// TIA Portal project "DrMartens2024_12_10_LMQTT_Client_V17" (V17)

(* hardware
DEVICE "S7-1200 station_1"  S7-1200 Station
   slot 0: "Rack_0"  S7-1200 Rack  Rack  V1.0
   slot 1: "MqttPlc1200"  CPU 1214C DC/DC/DC  6ES7 214-1AG40-0XB0  V4.4
DEVICE "S71500/ET200MP station_2"  S7-1500 station
   slot 0: "Rail_0"  Rack  6ES7 590-1***0-0AA0
   slot 1: "MqttPlc1500"  CPU 1517F-3 PN/DP  6ES7 517-3FP00-0AB0  V2.8
      slot 3: "CPU display_1"  6ES7591-1BA00-0AA0
      slot 32768: "PROFINET interface_1"  X1
         slot 32769: "Port_1"  X1 P1
         slot 32770: "Port_2"  X1 P2
      slot 33024: "PROFINET interface_2"  X2
      slot 33280: "DP interface_1"  X3
      slot 34817: "Virtual CP interface port_1"  Virtual CP interface port  Virtual CP interface port
*)

// ===== PLC "MqttPlc1200"  CPU 1214C DC/DC/DC =====

VAR_GLOBAL   // PLC tag table "Default tag table"
   "I0_0_Speed" AT %I0.0 : Bool;   // Speed - Sensor
   "I0_1_RunStop_Machine" AT %I0.1 : Bool;   // Relay
   "I0_2_Signal_Xilanh_Push" AT %I0.2 : Bool;   // Relay
   "I0_3_Signal_Pedal" AT %I0.3 : Bool;   // Relay: TRUE: Đi vào, FALSE : Đi ra
   "I0_4_RunStop_Inverter" AT %I0.4 : Bool;
   "I0_5_Spare" AT %I0.5 : Bool;
   "I0_6_Spare" AT %I0.6 : Bool;
   "I0_7_Spare" AT %I0.7 : Bool;
   "AI_Module_Ch00_Pressure_In" AT %IW96 : Int;   // Analog dòng
   "AI_Module_Ch01__Pressure_Out" AT %IW98 : Int;   // Analog spare
   "AI_Module_Ch02_Temperature" AT %IW100 : Int;   // Analog nhiệt độ
   "AI_Module_Ch03" AT %IW102 : Int;   // Analog Pressure Out
   "System_Byte" AT %MB1 : Byte;
   "FirstScan" AT %M1.0 : Bool;
   "DiagStatusUpdate" AT %M1.1 : Bool;
   "AlwaysTRUE" AT %M1.2 : Bool;
   "AlwaysFALSE" AT %M1.3 : Bool;
   "Clock_Byte" AT %MB0 : Byte;
   "Clock_10Hz" AT %M0.0 : Bool;
   "Clock_5Hz" AT %M0.1 : Bool;
   "Clock_2.5Hz" AT %M0.2 : Bool;
   "Clock_2Hz" AT %M0.3 : Bool;
   "Clock_1.25Hz" AT %M0.4 : Bool;
   "Clock_1Hz" AT %M0.5 : Bool;
   "Clock_0.625Hz" AT %M0.6 : Bool;
   "Clock_0.5Hz" AT %M0.7 : Bool;
   "M_Speed" AT %M100.0 : Bool;
   "M_RunStop_Machine" AT %M100.1 : Bool;
   "M_Xilanh_Push" AT %M100.2 : Bool;
   "M_Pedal" AT %M100.3 : Bool;
   "M_RunStop_Inverter" AT %M100.4 : Bool;
   "Input 5 Spare" AT %M100.5 : Bool;
   "Input 6 Spare" AT %M100.6 : Bool;
   "Input 7 Spare" AT %M100.7 : Bool;
   "M_Temperature" AT %MW4 : Int;
   "M_Current" AT %MW6 : Int;
   "M_AnalogPlc_Spare" AT %MW8 : Int;
   "M_Pressure Out" AT %MW16 : Int;
   "tag_idx" AT %MW18 : Int;
   "SignalP_RaisingCounter" AT %M200.0 : Bool;
   "SignalStatusMachineP" AT %M200.1 : Bool;
   "TagSignalStatusMachineP" AT %M200.2 : Bool;
   "TagSignalStatusMachineN" AT %M200.3 : Bool;
   "ClearDataBufferLossInShift" AT %M200.4 : Bool;
   "ClearDataBufferStatusMachineForServer" AT %M200.5 : Bool;
   "ClearSetDataDefaultLossGroupReason" AT %M200.6 : Bool;
   "PulseP_Check_ConnectHmi" AT %M200.7 : Bool;
   "Tag_1" AT %M500.0 : Bool;
   "Tag_2" AT %M601.0 : Bool;
   "Tag_3" AT %M601.2 : Bool;
   "Tag_4" AT %M600.4 : Bool;
   "Tag_5" AT %M700.0 : Bool;
   "Tag_6" AT %M700.1 : Bool;
   "Tag_7" AT %M700.2 : Bool;
   "AI_PLC_Ch00_Current" AT %IW64 : Int;   // AnalogPlcCh01
   "AI_PLC_Ch01" AT %IW66 : Int;   // AnalogPlcCh02
   "M_Pressure In" AT %MW20 : Int;
   "M_AnalogModule_Spare" AT %MW22 : Int;
   "Tag_8" AT %M201.0 : Bool;
   "Tag_9" AT %M202.1 : Bool;
   "Tag_10" AT %M303.0 : Bool;
   "Tag_11" AT %M303.2 : Bool;
   "Tag_12" AT %M303.1 : Bool;
   "Tag_13" AT %M404.0 : Bool;
   "Tag_14" AT %Q0.0 : Bool;
END_VAR

TYPE "SensorSimulation"
VERSION : 0.1
   STRUCT
      TimerTriggerON_x10ms : UInt := 100;   // Time-base x10ms
      TimerTriggerOFF_x10ms : UInt := 100;   // Time-base x10ms
      Output : Bool;
      nTempCounting : UInt;
   END_STRUCT;
END_TYPE

TYPE "DataShowChart"
VERSION : 0.1
   STRUCT
      Actual : DInt;
      Max : DInt;
      Min : DInt;
      AxisY_Max : DInt;
      AxisY_Min : DInt;
   END_STRUCT;
END_TYPE

TYPE "MachineEventDatatype"
VERSION : 0.1
   STRUCT
      id : UDInt;
      losscode : UInt;
      startTime : DTL;
      endTime : DTL;
      duration : UDInt;
      statusServer : USInt;   // 0: undefine; 1: stop; 2: run; 3: server-read; 4: server-updated
   END_STRUCT;
END_TYPE

TYPE "LossDescriptionDatatype"
VERSION : 0.1
   STRUCT
      description : String[30];
      group_id : UInt;
   END_STRUCT;
END_TYPE

TYPE "SpeedSensorType"
VERSION : 0.1
   STRUCT
      bStartCalculateSpeed : Bool;   // Bit lưu trạng thái vào quy trình đo speed
      TimeSpeed : Time;   // Time tính được giữa 2 lần interrupt
      idx : Int;   // Số lần tính speed
      "Out Current Speed" : Int;   // Tốc độ hiện tại đo được
   END_STRUCT;
END_TYPE

TYPE "AnalogSensorType"
VERSION : 0.1
   STRUCT
      MinRealScale : Real;   // 0V
      MaxRealScale : Real := 10.0;   // 10V
      real_Values : Array[0..3] of Real;   // Giá trị hiện tại dạng Real
      dint_Values : Array[0..3] of DInt;   // Giá trị hiện tại dạng Dint
      CurrentRealValue : Real;
      CurrentDintValue : DInt;
      digit : USInt;   // bao nhiêu số thập phân
   END_STRUCT;
END_TYPE

TYPE "MachineEventListView"
VERSION : 0.1
   STRUCT
      "no." : UInt;
      id : UDInt;
      LossCode : UInt;
      GroupLossReason : String[30];
      Description : String[30];
      StartDateAsStr : String[10];
      StartTimeAsStr : String[10];
      EndDateAsStr : String[10];
      EndTimeAsStr : String[10];
      DurationAsStr : String[12];
      StatusServer : UInt;   // 0: undefine; 1: stop; 2: run; 3: server-read; 4: server-updated
      IsHaveData : Bool;
   END_STRUCT;
END_TYPE

TYPE "Setting_CommonSensor"
VERSION : 0.1
   STRUCT
      "RangMinSensor(x100)" : DInt;   // Giá trị min của cảm biến
      "RangMaxSensor(x100)" : DInt;   // Giá trị max của cảm biến
      "Offset(x100)" : DInt;
      "SettingLower(x100)" : DInt;   // Cài đặt cận dưới
      "SettingUpper(x100)" : DInt;   // Cài đặt cận trên
   END_STRUCT;
END_TYPE

TYPE "Setting_WheelSpeed"
VERSION : 0.1
   STRUCT
      "Offset(x100)" : DInt;
      "SettingLower(x100)" : DInt;   // Cài đặt cận dưới
      "SettingUpper(x100)" : DInt;   // Cài đặt cận trên
      "GearRatio(x100)" : UInt;
      NumberOfGears : UInt;
   END_STRUCT;
END_TYPE

TYPE "Setting_ForceXilanh"
VERSION : 0.1
   STRUCT
      "Offset(x100)" : DInt;
      "SettingLower(x100)" : DInt;   // Cài đặt cận dưới
      "SettingUpper(x100)" : DInt;   // Cài đặt cận trên
      "Area(cm2 x 100)" : UInt;
      "CoefficientUnit(x100)" : DInt;
   END_STRUCT;
END_TYPE

TYPE "InforPage"
VERSION : 0.1
   STRUCT
      TotalData : UDInt := 0;
      MaxPage : UDInt := 1;
      PageCurrent : UDInt := 1;
   END_STRUCT;
END_TYPE

TYPE "HMI_Sensor_CommonSensor"
VERSION : 0.1
   STRUCT
      Common : "Setting_CommonSensor";
      "ValueActual(x100)" : DInt;
      "ValueActualContainOffset(x100)" : DInt;
      Alarm : UInt;
      AnalogActual : Int;
   END_STRUCT;
END_TYPE

TYPE "InforStation"
VERSION : 0.1
   STRUCT
      Factory : String[30];
      Workshop : String[30];
      LineName : String[30];
      MachineName : String[30];
      MachineCode : String[10];
   END_STRUCT;
END_TYPE

TYPE "StatusMachineBuffer"
VERSION : 0.1
   STRUCT
      time_start : DTL;
      timer_end : DTL;
      status : USInt;   // 0:Undefine 1: Run, 2: Idle, 3: Stop, 4:Offline
   END_STRUCT;
END_TYPE

TYPE "InforSensor"
VERSION : 0.1
   STRUCT
      "CurrentNotOffset(x100)" : DInt;
      "Current(x100)" : DInt;
      "Upper(x100)" : DInt;
      "Lower(x100)" : DInt;
      AnalogCurrent : DInt;
      "Offset(x100)" : DInt;
      "RangeMinSensor(x100)" : DInt;
      "RangeMaxSensor(x100)" : DInt;
      Alarm : UInt;
   END_STRUCT;
END_TYPE

TYPE "SettingWheelSpeed"
VERSION : 0.1
   STRUCT
      Infor : "InforSensor";
      "GearRatio(x100)" : UInt;
      NumberOfGears : UInt;
   END_STRUCT;
END_TYPE

TYPE "SettingForce"
VERSION : 0.1
   STRUCT
      Infor : "InforSensor";
      Area : UInt;
      "CoefficientUnit(x100)" : DInt;
   END_STRUCT;
END_TYPE

TYPE "SearchLoss"
VERSION : 0.1
   STRUCT
      Year : UInt;
      Month : UInt;
      Day : UInt;
   END_STRUCT;
END_TYPE

TYPE "SparePart"
VERSION : 0.1
   STRUCT
      "name" : String[30];
      product_count : UDInt;
      start_time : DTL;
      end_time : DTL;
   END_STRUCT;
END_TYPE

TYPE "change_setting"
VERSION : 0.1
   STRUCT
      confirm : Bool;
      cancel : Bool;
   END_STRUCT;
END_TYPE

TYPE "SparePartHMI"
VERSION : 0.1
   STRUCT
      "No." : UDInt;
      ProductCount : UDInt;
      IsHaveData : Bool;
      "Name" : String[30];
      StartTime : String[20];
      EndTime : String[20];
   END_STRUCT;
END_TYPE

TYPE "HMI_WheelSpeed"
VERSION : 0.1
   STRUCT
      Common : "Setting_WheelSpeed";
      "ValueActual(x100)" : DInt;
      "ValueActualContainOffset(x100)" : DInt;
      "SpeedMeasure(x100)" : DInt;
      Alarm : UInt;
   END_STRUCT;
END_TYPE

TYPE "HMI_ForceXilanh"
VERSION : 0.1
   STRUCT
      Common : "Setting_ForceXilanh";
      "ValueActual(x100)" : DInt;
      "ValueActualContainOffset(x100)" : DInt;
      Alarm : UInt;
   END_STRUCT;
END_TYPE

TYPE "SortBuffer"
VERSION : 0.1
   STRUCT
      id : UDInt;
      index_buffer : UInt;
   END_STRUCT;
END_TYPE

TYPE "ReasonLossHmi"
VERSION : 0.1
   STRUCT
      description : String[30];
      group_id : UInt;
      index_buffer : UInt;
   END_STRUCT;
END_TYPE

// folder: Common

TYPE "typeDiagnostics"
TITLE = typeDiagnostics
VERSION : 0.1
// Provides a structure for detailed diagnostics
   STRUCT
      status : Word;   // Status of the block or error identification when error occurred
      subfunctionStatus : DWord;   // Status or return value of called FBs, FCs and system blocks
      stateNumber : DInt;   // State in the state machine of the block where the error occurred
   END_STRUCT;
END_TYPE

// folder: LMQTT

TYPE "LMQTT_typeConnParam"
TITLE = LMQTT_typeConnParams
VERSION : 0.1
// Specifies connection parameters for the mqtt connection
   STRUCT
      hwId : Hw_Any;   // Hardware identifier of the interface. 0: interface is selected automatically
      connId : Conn_Ouc := 1;   // Unique connection identifier (1..4095)
      broker : String;   // Hostname or IP address of broker
      port : UInt := 1883;   // Port on the broker
      tls : Struct   // Parameters for TLS encryption
         enableTls : Bool;   // TRUE: Enables TLS, FALSE: disable TLS
         validateServerIdentity : Bool;   // TRUE: Validate server certificate, FALSE: No validation of server certificate
         brokerCert : UDInt;   // ID of the broker's certificate in TIA Portal
         clientCert : UDInt;   // ID of the client's certificate in TIA Portal
      END_STRUCT;
      keepAlive : UInt;   // Keepalive mechanism for MQTT in seconds. 0: disabled.
   END_STRUCT;
END_TYPE

// folder: (top level)

DATA_BLOCK "InstLMQTT_Client"   // DB1
{ S7_Optimized_Access := 'TRUE' }
AUTHOR : SiemensAG
FAMILY : MQTT
VERSION : 1.0
// stored: InstanceOfName LMQTT_Client
"LMQTT_Client"
BEGIN
END_DATA_BLOCK

DATA_BLOCK "MqttDb"   // DB2
TITLE = Configuration Data block example for LMQTT_Client
{ S7_Optimized_Access := 'TRUE' }
AUTHOR : Siemens
FAMILY : LMQTT
VERSION : 1.0
// This block is an example how to control the LMQTT_Client function block
   VAR
      control : Struct   // Input of the FB
         enable : Bool;   // Set TRUE, to establish a connection - set to FALSE to disconnect
         publish : Bool;   // Rising Edge: Sends a message
         subscribe : Bool;   // Rising Edge: Subscribes to a topic
         unsubscribe : Bool;   // Rising Edge: Unsubscribes to a topic
      END_STRUCT;
      output : Struct   // Output Information of the FB
         valid : Bool;   // TRUE: Valid set of output values available at the FB
         done : Bool;   // TRUE: If last Request was successfull
         busy : Bool;   // TRUE: FB is not finished and new output values can be expected
         error : Bool;   // TRUE: An error occurred during the execution of the FB
         status : Word;   // 16#0000 - 16#7FFF: Status of the FB, 16#8000 - 16#FFFF: Error identification
         diagnostics : "typeDiagnostics";   // Diagnostics information of FB (optional)
      END_STRUCT;
      connParam : "LMQTT_typeConnParam";   // Connection Parameters
      clientIdentifier : WString[20] := WSTRING#'abcd123';   // ClientId with one or more characters
      username : WString[20] := WSTRING#'uehmqtt_passthedung';   // Username used for connect
      password : WString[20] := WSTRING#'uehmqtt_passthedung';   // Password used for connect
      willTopic : WString[20];   // Topic where the last will message is sent
      willMsgPayload : Array[0..99] of Byte;   // Last will message Data - valid bytes in this array must be written in input 'willMsgLen'
      willMsgLen : UInt;   // Valid number of elements in Will Message Data Array. Max 65535 Byte allowed by MQTT Spec.
      qos : USInt;   // Sets QoS 0,1 or 2 for the Publish and Will Message - Subscribe only allows QoS 0 and 1
      mqttTopic : WString[100] := WSTRING#'martens';   // Mqtt Topic to Publish / Subscribe / Unsubscribe
      publishMsgPayload : Array[0..999] of Byte;   // Message Data to Publish - valid bytes in this array must be written in input 'publishMsgLen'
      publishMsgLen : UDInt := 5;   // Valid number of elements in publish message data Array
      retain : Bool;   // TRUE: Published Message will be set to retain on MQTT broker
      receivedTopic : WString[200];   // Mqtt Topic of received message
      receivedMsgPayload : Array[0..999] of Byte;   // Mqtt message data that was received - valid bytes in this array indicated by 'receivedMsgDataLen' output
      receivedMsgDataLen : UDInt;   // Amount of Bytes received in receivedMessage INOUT area
      receivedMsgStatus : USInt;   // 0: No new Message, 1: New valid Message received and available at InOut area, 2: New message, but data is invalid (wrong message len or message could not be copied to InOut received topic or received message)
   END_VAR
BEGIN
   willMsgPayload[0] := 16#6F;
   willMsgPayload[1] := 16#66;
   willMsgPayload[2] := 16#66;
   willMsgPayload[3] := 16#6C;
   willMsgPayload[4] := 16#69;
   willMsgPayload[5] := 16#6E;
   willMsgPayload[6] := 16#65;
   publishMsgPayload[1] := 16#65;
   publishMsgPayload[2] := 16#6c;
   publishMsgPayload[3] := 16#6c;
   publishMsgPayload[4] := 16#6f;
   publishMsgPayload[5] := 16#20;
   publishMsgPayload[6] := 16#77;
   publishMsgPayload[7] := 16#6f;
   publishMsgPayload[8] := 16#72;
   publishMsgPayload[9] := 16#6c;
   publishMsgPayload[10] := 16#64;
   publishMsgPayload[0] := 16#68;
   connParam.broker := '192.168.2.101';
END_DATA_BLOCK

DATA_BLOCK "1.2 Speed_Sensor_DB_1"   // DB9
{ S7_Optimized_Access := 'TRUE' }
VERSION : 0.1
// stored: InstanceOfName 1.2 Speed_Sensor
"1.2 Speed_Sensor"
BEGIN
END_DATA_BLOCK

DATA_BLOCK "CounterFB_DB"   // DB12
{ S7_Optimized_Access := 'TRUE' }
VERSION : 0.1
// stored: InstanceOfName CounterFB
"CounterFB"
BEGIN
END_DATA_BLOCK

DATA_BLOCK "DB_Machine"   // DB14
{ S7_Optimized_Access := 'TRUE' }
VERSION : 0.1
   VAR RETAIN
      "product counter" : UDInt;
      AnalogSensorMax : Int := 27648;
      AnalogSensorMin : Int := 0;
      machine_run : Bool;   // Máy chạy/dừng
      machine_total_runtime : String[20];
      machine_total_stoptime : String[20];
      system_alarm : Bool;   // Bit báo đang có alarms
      system_alarm_description : String[40];
      machine_event_total_page : USInt;
      CounterTemp : UDInt;
      CounterMachineInShift : UDInt;
      CounterRaw : UDInt;   // Không Rs qua ca
      MachineStatus : UInt;   // 1: Run, 2: Stop, 3: Idle
      MachineStatusPrevious : UInt;
      EventReloadPageAssignLossInShift : USInt := 1;   // 1: Có Loss, 2 PLC rs
      PageCurrentServerSparePartPrevious : UDInt;
      PageCurrentServerHistoricalPrevious : UDInt;
      NumberLossInShift : UDInt;
   END_VAR
   VAR
      CounterSpeed : UInt;
      value_temp : "SortBuffer";
      buffer_index_sort : Array[1..100] of "SortBuffer";
      SpeedMeasure : DInt;
      SpeedMotor : DInt;
      Test001 : DInt;
   END_VAR
   VAR RETAIN
      PageLossInShiftHmiPrevious : UDInt;
      PageHistoricalHmiPrevious : UDInt;
      PageHistoricalServerPrevious : UDInt;
   END_VAR
BEGIN
END_DATA_BLOCK

DATA_BLOCK "StartStop_DB"   // DB16
{ S7_Optimized_Access := 'TRUE' }
VERSION : 0.1
// stored: InstanceOfName StartStop
"StartStop"
BEGIN
END_DATA_BLOCK

DATA_BLOCK "TagTest"   // DB17
{ S7_Optimized_Access := 'TRUE' }
VERSION : 0.1
   VAR
      Test1 : UInt;
      Test2 : UInt;
      Test3 : UInt;
      AnalogTemperature : Int;
      AnalogCurrent : Int;
      AnalogPressure : Int;
      TestRandomSparePart : Bool;
      TestRandomHistorical : Bool;
      Speed1 : DInt;
      Speed2 : DInt;
      TestPulse : UInt;
      Pulse : UInt;
      CounterSpeed : UInt;
      SpeedActual_2 : DInt;
      SpeedActualContainOffset_2 : DInt;
      Test01 : DInt;
      MoveSparePart : Bool;
      IndexUpdateLossServer : USInt;
      NumberOnPowerPLC : UInt;
      NumberServerResetCounter : UInt;
   END_VAR
   VAR RETAIN
      TimeLastOnPlcRealTime : DTL;
      TimeLastOnPlc : DTL;
   END_VAR
BEGIN
END_DATA_BLOCK

DATA_BLOCK "DB_DataHMI"   // DB18
{ S7_Optimized_Access := 'FALSE' }
VERSION : 0.1
   VAR
      CounterCurrent : UDInt;
      MachineStatus : UInt;   // 1: Run, 2: Stop, 3 Sand By, NG
      TypeLayer : UInt := 1;   // 1: 1 layer, 2: 2 layer
      DataLossHistoricalShowHmiDTO : Array[1..5] of "MachineEventListView";
      PageDataLossHistorical : "InforPage";
      SearchDataLoss : "SearchLoss";
      ActionSearchLossHistorical : Bool;
      TotalTimeLossHistorical : String[20];
      TotalDataHistorical : UDInt;
      SwicthPageLossHistorical : UInt;   // 1: Tăng, 2: Giảm, 3. PLC Reset, NG
      DataLossInShiftShowHmiDTO : Array[1..5] of "MachineEventListView";
      PageDataLossInShift : "InforPage";
      TotalDataInShift : UDInt;
      SwitchTabPageLossInShift : UInt;   // 1: Tăng, 2: Giảm, 3. PLC Reset, NG
      EventSwitchPageLossInShift : Bool;
      PageDataLossReason : "InforPage";
      SwitchTabPageLossReason : UInt;   // 1: Tăng, 2: Giảm, 3. PLC Reset, NG
      NumberRowEachPage : UInt;
      LossGroupHmiDTO : Array[1..10] of String[30];
      LossDescriptionHmiDTO : Array[1..10] of "ReasonLossHmi";
      EventCheckLossGroup : UInt;   // 1: Yêu cầu PLC Update, 2 PLC Rs, NG
      LossGroupSelectId : UInt;   // Value: 1->10
      CheckboxLossGroup : Array[1..10] of UInt;
      VisibleCheckboxLossGroup : Array[1..10] of Bool;
      EventCheckLossReason : UInt;   // 1: Yêu cầu PLC Update, 2 PLC Rs, NG
      LossReasonSelectId : UInt;   // Value: 1->10
      CheckboxLossReason : Array[1..10] of UInt;
      VisibleCheckboxLossReason : Array[1..10] of Bool;
      EventIndexRowInShift : Array[1..5] of Bool;   // Từ 1 đến 5
      EventIndexRowHistorical : Array[1..5] of Bool;
      IndexRowAssignLoss : UInt;
      TypeAssignLoss : UInt;   // 1: In Shift, 2: Historical, 3: Loss Over Time
      StartTimeAssignLossCurrent : String[20];
      EndTimeAssignLossCurrent : String[20];
      DurationAssignLossCurrent : String[20];
      TextLossGroupAssignLossCurrent : String[30];
      TextLossReasonAssignLossCurrent : String[30];
      ActionAssignLossInShift : Bool;   // 1 Request, 2 PLC Rs
      ActionAssignLossHistorical : Bool;
      CancelAssignLoss : Bool;
      InforStation : "InforStation";
      "CounterFilterOn(ms)" : UInt;
      "CounterFilterOff(ms)" : UInt;
      "TimeThresholdLoss(ms)" : UInt;
      "TimeThresholdClearBlade(ms)" : UInt;
      "TimeThresholdShowWarningAssignLoss(s)" : UInt;
      AnalogSensorMin : DInt;
      AnalogSensorMax : DInt;
      IO_Digital : Array[1..16] of Bool;
      PageHomeStartTimeStatusCurrent : String[20];
      PageHomeEndTimeStatusCurrent : String[20];
      PageHomeDurationStatusCurrent : String[10];
      PageHomeBitShowAssignLoss : Bool;
      FlagCancelAssignLossCurrent : Bool;   // Cờ này dùng để ẩn assignloss hiện tại nếu bấm cancel, đợi qua los mới mới về false
      EventAssignLossCurrent : Bool;
      StatusConnectController : Bool;   // 1: Connected, 2 Disconnect
      StatusConnectServer : Bool;   // 1: Connected, 2 Disconnect
      DataSparePartShowHmiDTO : Array[1..5] of "SparePartHMI";
      PageDataSparePart : "InforPage";
      SwitchPageSparePart : UInt;   // 1: Tăng, 2: Giảm, 3. PLC Reset, NG
      ActionSearchLossSparePart : Bool;
      ActionRefreshLossSparePart : Bool;
      DataChartSpeed : "DataShowChart";
      DataChartCurrent : "DataShowChart";
      DataChartBladeTemperature : "DataShowChart";
      DataChartPressureOut : "DataShowChart";
      EventBitShowNoDataHistorical : Bool;
      EventBitShowSaveSettingSuccess : Bool;
      BladeTemperature : "HMI_Sensor_CommonSensor";
      Current : "HMI_Sensor_CommonSensor";
      PressureIn : "HMI_Sensor_CommonSensor";
      PressureOut : "HMI_Sensor_CommonSensor";
      "ValuePressureOut_MPa(x100)" : DInt;
      WheelSpeed : "HMI_WheelSpeed";
      "TimePerPulseSensorSpeed(x1ms)" : DInt;
      ForceXilanh : "HMI_ForceXilanh";
      ActionConfirmSetting : Bool;
      ActionCancelSetting : Bool;
      ActionRefreshLossInShift : Bool;
      IndexTabSetting : Int;   // 1: Information, 2 General, 3 BladeTemp, 4 Current,5 WheelSpeed,6 Force
      BitReloadSettingToHMI : Bool;
      EventChangePageLossInShift : Bool;
      DataFloatWrite : Real;
      DataFloatRead : Real;
      RequestLoadGroupReasonLoss : Bool;
      EventBitShowPopupLoading : Bool;
      EventBitShowPopupErrorFormatDaySearch : Bool;
      Second_HMI : Int;
      Minute_HMI : Int;
      Hour_HMI : Int;
      Day_HMI : Int;
      Month_HMI : Int;
      Year_HMI : Int;
   END_VAR
BEGIN
   PageDataLossHistorical.PageCurrent := 1;
   PageDataLossHistorical.MaxPage := 1;
   PageDataSparePart.MaxPage := 1;
   PageDataSparePart.PageCurrent := 1;
END_DATA_BLOCK

DATA_BLOCK "Speed_Sensor_DB_Speed_Average"   // DB19
{ S7_Optimized_Access := 'TRUE' }
VERSION : 0.1
// stored: InstanceOfName Speed_Sensor
"Speed_Sensor"
BEGIN
END_DATA_BLOCK

DATA_BLOCK "StatusMachine_DB"   // DB20
{ S7_Optimized_Access := 'TRUE' }
VERSION : 0.1
// stored: InstanceOfName StatusMachine
"StatusMachine"
BEGIN
END_DATA_BLOCK

DATA_BLOCK "StatusMachineSendServerDB"   // DB23
{ S7_Optimized_Access := 'FALSE' }
VERSION : 0.1
   VAR
      StatusMachineBuffer : Array[1..50] of "StatusMachineBuffer";
      index_current : USInt := 1;
      min_index_buffer : USInt := 1;
      max_index_buffer : USInt := 50;
   END_VAR
BEGIN
END_DATA_BLOCK

DATA_BLOCK "DataSetting"   // DB24
{ S7_Optimized_Access := 'FALSE' }
VERSION : 0.1
   VAR
      InforStation : "InforStation";
      "CounterFilterOn(ms)" : UInt;
      "CounterFilterOff(ms)" : UInt;
      "TimeThresholdLoss(ms)" : UInt;
      "TimeThresholdClearBlade(ms)" : UInt;
      "TimeThresholdShowWarningAssignLoss(s)" : UInt;
      SettingBladeTemp : "Setting_CommonSensor";
      SettingCurrent : "Setting_CommonSensor";
      SettingPresureIn : "Setting_CommonSensor";
      SettingPresureOut : "Setting_CommonSensor";
      SettingWheelSpeed : "Setting_WheelSpeed";
      SettingForceXilanh : "Setting_ForceXilanh";
      TypeLayer : UInt;   // 1: 1 layer, 2: 2 layer
   END_VAR
BEGIN
   InforStation.MachineCode := 'machine1';
   InforStation.Factory := 'Factory1';
   InforStation.Workshop := 'Workshop1';
   InforStation.LineName := 'Line1';
END_DATA_BLOCK

DATA_BLOCK "CheckConnectPLCServer_DB"   // DB25
{ S7_Optimized_Access := 'TRUE' }
VERSION : 0.1
// stored: InstanceOfName CheckConnectPLCServer
"CheckConnectPLCServer"
BEGIN
END_DATA_BLOCK

DATA_BLOCK "CreatePulse_DB_1_Simulation_Signal_Speed"   // DB27
{ S7_Optimized_Access := 'TRUE' }
VERSION : 0.1
// stored: InstanceOfName CreatePulse
"CreatePulse"
BEGIN
END_DATA_BLOCK

DATA_BLOCK "CreatePulse_DB_CheckConnectHMI"   // DB28
{ S7_Optimized_Access := 'TRUE' }
VERSION : 0.1
// stored: InstanceOfName CreatePulse
"CreatePulse"
BEGIN
END_DATA_BLOCK

DATA_BLOCK "CreatePulse_DB"   // DB29
{ S7_Optimized_Access := 'TRUE' }
VERSION : 0.1
// stored: InstanceOfName CreatePulse
"CreatePulse"
BEGIN
END_DATA_BLOCK

DATA_BLOCK "CreatePulse_DB_Update_Speed"   // DB30
{ S7_Optimized_Access := 'TRUE' }
VERSION : 0.1
// stored: InstanceOfName CreatePulse
"CreatePulse"
BEGIN
END_DATA_BLOCK

// folder: LossManagement

DATA_BLOCK "GLobalDB_LossManagementDB"   // DB11
{ S7_Optimized_Access := 'TRUE' }
VERSION : 0.1
   VAR RETAIN
      currentId : USInt := 1;
      startIdx : USInt := 1;
      endIdx : USInt := 100;
      total_run_time : UDInt;
      total_stop_time : UDInt;
      current_status_machine : "MachineEventDatatype";
      id_loss : UDInt := 1;
      index_buffer_loss_in_shift_current : USInt := 1;
   END_VAR
   VAR
      "duration_status_curent(ms)" : UDInt;
   END_VAR
BEGIN
END_DATA_BLOCK

DATA_BLOCK "SettingsDB_LossDescription"   // DB13
{ S7_Optimized_Access := 'FALSE' }
VERSION : 0.1
   VAR
      loss_name_group : Array[1..10] of String[30];
      loss_descriptions : Array[1..100] of "LossDescriptionDatatype";
      number_loss_reason : USInt;
   END_VAR
BEGIN
   loss_descriptions[1].description := 'Unassign loss';
   loss_descriptions[2].description := 'loss code 2';
   loss_descriptions[3].description := 'loss code 3';
   loss_descriptions[4].description := 'loss code 4';
   loss_descriptions[5].description := 'loss code 5';
   loss_descriptions[6].description := 'loss code 6';
   loss_descriptions[7].description := 'loss code 7';
   loss_descriptions[8].description := 'loss code 8';
   loss_descriptions[9].description := 'loss code 9';
   loss_descriptions[10].description := 'loss code 10';
   loss_descriptions[11].description := 'loss code 11';
   loss_descriptions[12].description := 'loss code 12';
   loss_descriptions[13].description := 'loss code 13';
   loss_descriptions[14].description := 'loss code 14';
   loss_descriptions[15].description := 'loss code 15';
   loss_descriptions[16].description := 'loss code 16';
   loss_descriptions[17].description := 'loss code 17';
   loss_descriptions[18].description := 'loss code 18';
   loss_descriptions[19].description := 'loss code 19';
   loss_descriptions[20].description := 'loss code 20';
   loss_descriptions[21].description := 'loss code 21';
   loss_descriptions[22].description := 'loss code 22';
   loss_descriptions[23].description := 'loss code 23';
   loss_descriptions[24].description := 'loss code 24';
   loss_descriptions[25].description := 'loss code 25';
   loss_descriptions[26].description := 'loss code 26';
   loss_descriptions[27].description := 'loss code 27';
   loss_descriptions[28].description := 'loss code 28';
   loss_descriptions[29].description := 'loss code 29';
   loss_descriptions[30].description := 'loss code 30';
END_DATA_BLOCK

DATA_BLOCK "BuffersLoss_DB"   // DB15
{ S7_Optimized_Access := 'FALSE' }
VERSION : 0.1
   VAR
      buffer_loss_in_shift : Array[1..100] of "MachineEventDatatype";
      buffer_loss_in_historical : Array[1..50] of "MachineEventDatatype";
   END_VAR
BEGIN
END_DATA_BLOCK

DATA_BLOCK "BufferServerSend"   // DB22
{ S7_Optimized_Access := 'FALSE' }
VERSION : 0.1
   VAR
      buffer_spare_part : Array[1..30] of "SparePart";
   END_VAR
BEGIN
END_DATA_BLOCK

// folder: RTC

DATA_BLOCK "GlobalDB_RTC"   // DB10
{ S7_Optimized_Access := 'TRUE' }
VERSION : 0.1
   VAR
      RTC_Local : DTL;
      Status : Int;
      RTC_System : DTL;
      RTC_UTC : USInt;
      GetStatus : Int;
      SetStatus : Int;
      RTC_Defaul : DTL;   // Thời gian set defaul, mặc định xóa
   END_VAR
BEGIN
END_DATA_BLOCK

// folder: Sensor-Speed

DATA_BLOCK "SensorSpeed_DB"   // DB5
{ S7_Optimized_Access := 'TRUE' }
VERSION : 0.1
   VAR
      "speed sensor" : "SpeedSensorType";
      array_speed_temp : Array[1..50] of Real;
      index_array_speed : USInt;
   END_VAR
BEGIN
END_DATA_BLOCK

// folder: Sensor-Speed/Data

DATA_BLOCK "1.2 Speed_Sensor_DB"   // DB3
{ S7_Optimized_Access := 'TRUE' }
VERSION : 0.1
// stored: InstanceOfName 1.2 Speed_Sensor
"1.2 Speed_Sensor"
BEGIN
END_DATA_BLOCK

DATA_BLOCK "1.3 Interrupt_DB"   // DB4
{ S7_Optimized_Access := 'TRUE' }
VERSION : 0.1
// stored: InstanceOfName 1.3 Speed Interrupt
"1.3 Speed Interrupt"
BEGIN
END_DATA_BLOCK

// folder: Sensor-StartStop

DATA_BLOCK "InputFilter_DB_1"   // DB8
{ S7_Optimized_Access := 'TRUE' }
VERSION : 0.1
// stored: InstanceOfName InputFilter
"InputFilter"
BEGIN
END_DATA_BLOCK

// folder: Server

DATA_BLOCK "Analogs_DB"   // DB7
{ S7_Optimized_Access := 'TRUE' }
VERSION : 0.1
   VAR RETAIN
      Temperature : "AnalogSensorType";   // Nhiệt độ
      Current : "AnalogSensorType";   // Dòng điện
      Pressure_IN : "AnalogSensorType";   // Áp suất vào
      Pressure_OUT : "AnalogSensorType";   // Áp suất ra
   END_VAR
BEGIN
END_DATA_BLOCK

DATA_BLOCK "DB_Server"   // DB21
{ S7_Optimized_Access := 'FALSE' }
VERSION : 0.1
   VAR
      InforStation : "InforStation";
      "CounterFilterOn(ms)" : UInt;
      "CounterFilterOff(ms)" : UInt;
      "TimeThresholdLoss(ms)" : UInt;
      "TimeThresholdShowWarningAssignLoss(s)" : UInt;
      SettingBladeTemp : "InforSensor";
      SettingCurrent : "InforSensor";
      SettingWheelSpeed : "SettingWheelSpeed";
      SettingForce : "SettingForce";
      SensorPresureIn : "InforSensor";
      SensorPresureOut : "InforSensor";
      SyncSettings : USInt;   // 1: HMI có thay đổi, 2: Server có thay đổi, 3: Done Sync
      RequestServerWriteLossGroup_Reason : USInt;   // 1 Request, 2 Server Rs, NG
      RequestServerUpdateLossInShift : USInt;   // 1 Request, 2 Server Rs, NG
      RequestServerUpdateLossHistorical : USInt;   // 1 Request, 2 Server Rs, NG
      MachineStatus : SInt;
      CounterMachineInShift : UDInt;
      CounterRaw : UDInt;
      TypeLayer : UInt := 1;   // 1: 1 layer, 2: 2 layer
      StartTimeStatusCurrent : DTL;
      EndTimeStatusCurrent : DTL;
      DurationStatusCurrent : UDInt;
      ConnectPLC : Bool;
      PageHistorical : "InforPage";
      SearchDataLossHistorical : "SearchLoss";
      ActionSearchLossHistorical : UInt;   // 1 Request, 2 Server Rs, 3 PLC Rs 4 Format DateTime sai
      PageDataSparePart : "InforPage";   // 1: Server gửi data, 2 Plc Rs, 3 Done, NG
      ActionSearchLossSparePart : UInt;
      RequestServerUpdateBufferStatusMachine : USInt;   // 1 Request, 2 Server Rs, NG
      TotalDurationPageHistorical : UDInt;
      LossInShiftAssign : "MachineEventDatatype";   // Thời gian bắt đầu Loss Assign trên Server
      RealTimeFromPC : DTL;
      SyncTimeFromPC : Bool;
      "TimeThresholdBlade(ms)" : UInt;
      EventResetCounterInShift : Bool;
   END_VAR
BEGIN
   PageDataSparePart.MaxPage := 1;
   PageDataSparePart.PageCurrent := 1;
END_DATA_BLOCK

// folder: Simulation

DATA_BLOCK "GlobalDB_Simulation"   // DB6
{ S7_Optimized_Access := 'TRUE' }
VERSION : 0.1
   VAR
      SpeedSensors : Array[0..10] of "SensorSimulation";
      CounterSensors : Array[0..10] of "SensorSimulation";
   END_VAR
BEGIN
END_DATA_BLOCK

DATA_BLOCK "RandomAnalogs"   // DB26
{ S7_Optimized_Access := 'TRUE' }
VERSION : 0.1
   VAR
      Speed_Value : Int;
      Temp_Analog : Int;
      Pressure_Analog : Int;
      Current_Analog : Int;
      IndexRandom : USInt;
      ValueTemp : Int;
      from_random : Int;
      to_random : Int;
   END_VAR
BEGIN
END_DATA_BLOCK

// folder: (top level)

FUNCTION_BLOCK "StatusMachine"   // FB7, LAD
{ S7_Optimized_Access := 'TRUE' }
VERSION : 0.1
   VAR_INPUT
      SignalMachine : Bool;
      SignalInverter : Bool;
      "SignalXilanh(true: push)" : Bool;
      TimeOutRunToIdle : UDInt;
      TimeOutClearBlade : UDInt;
   END_VAR
   VAR_OUTPUT
      Status : UInt;   // 1: Running, 2: Stop, 3: Idle, NG
   END_VAR
   VAR
      bTimeOutOperation : Bool;
      bTimeOutClearBlade : Bool;
      signal_xilanh_push_P : Bool;
      signal_xilanh_push_N : Bool;
      FlagXilanhPush : Bool;
      FlagXilanhPull : Bool;
      IEC_Timer_0_Instance : TON_TIME;
      IEC_Timer_0_Instance_Clear_Blade : TON_TIME;
   END_VAR
   VAR_TEMP
      TimeOperation : Time;
      TimeClearBlade : Time;
   END_VAR
   VAR CONSTANT
      "ThresholdIdle(x1ms)" : Int := 30000;
   END_VAR
   VAR_TEMP   // added for the SCL form of the ladder/FBD networks
      _w1 : Bool;
      _w2 : Bool;
   END_VAR
BEGIN

REGION Network 1: Case 1: Machine Stop
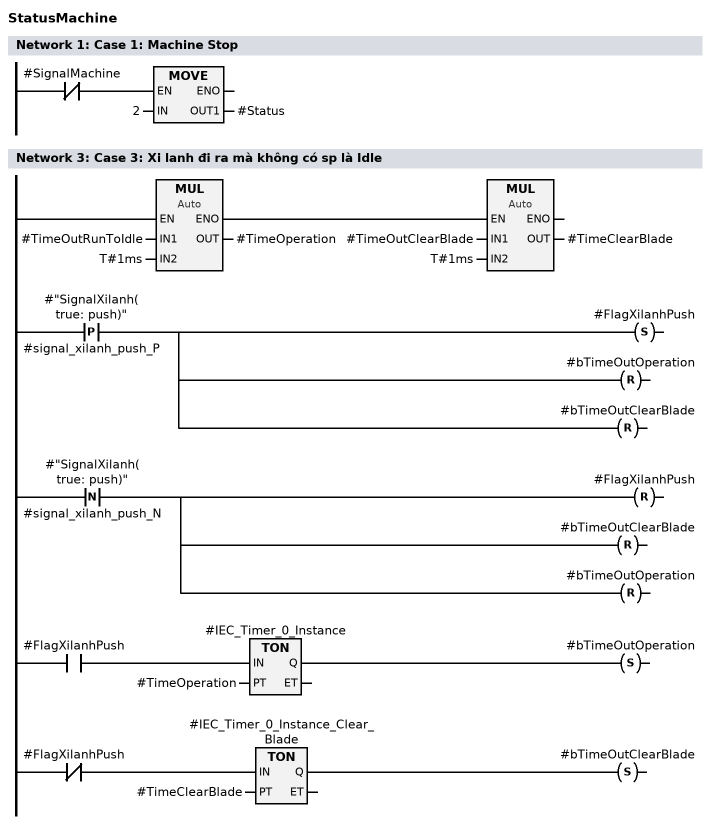
   RUNG wire#powerrail
      I_Contact( #SignalMachine )
      Move(in := 2, out1 => #Status)
   END_RUNG
   // the same network as SCL:
   IF NOT #SignalMachine THEN #Status := 2; END_IF;
END_REGION

REGION Network 2 (SCL): Case 2: Machine Run
   IF #SignalMachine=TRUE THEN
       IF #SignalInverter=TRUE  THEN
           IF #bTimeOutOperation = TRUE OR #bTimeOutClearBlade = TRUE THEN
               #Status := 3;
           ELSE
               #Status := 1;
           END_IF;
       ELSE
           #Status := 3;
       END_IF;
   END_IF;
END_REGION

REGION Network 3: Case 3: Xi lanh đi ra mà không có sp là Idle
   #TimeOperation := #TimeOutRunToIdle * T#1ms;
   #TimeClearBlade := #TimeOutClearBlade * T#1ms;
   #_w1 := #"SignalXilanh(true: push)" AND NOT #signal_xilanh_push_P;   // rising edge of #"SignalXilanh(true: push)"
   #signal_xilanh_push_P := #"SignalXilanh(true: push)";
   IF #_w1 THEN
       #FlagXilanhPush := TRUE;
       #bTimeOutOperation := FALSE;
       #bTimeOutClearBlade := FALSE;
   END_IF;
   #_w2 := NOT #"SignalXilanh(true: push)" AND #signal_xilanh_push_N;   // falling edge of #"SignalXilanh(true: push)"
   #signal_xilanh_push_N := #"SignalXilanh(true: push)";
   IF #_w2 THEN
       #FlagXilanhPush := FALSE;
       #bTimeOutClearBlade := FALSE;
       #bTimeOutOperation := FALSE;
   END_IF;
   #IEC_Timer_0_Instance(IN := #FlagXilanhPush, PT := #TimeOperation);   // TON
   IF #IEC_Timer_0_Instance.Q THEN #bTimeOutOperation := TRUE; END_IF;
   #IEC_Timer_0_Instance_Clear_Blade(IN := NOT #FlagXilanhPush, PT := #TimeClearBlade);   // TON
   IF #IEC_Timer_0_Instance_Clear_Blade.Q THEN #bTimeOutClearBlade := TRUE; END_IF;
END_REGION
END_FUNCTION_BLOCK

FUNCTION "CheckCalculatorCounter" : Void   // FC18, SCL
{ S7_Optimized_Access := 'TRUE' }
VERSION : 0.1
   VAR_INPUT
      TypeLayer : UInt;   // 1: 1 Layer, 2: 2 Layer
   END_VAR
   VAR_IN_OUT
      CounterTemp : UDInt;
   END_VAR
   VAR_TEMP
      Quotient : UDInt;
   END_VAR
BEGIN
   #Quotient := 0;
   IF #TypeLayer = 1 THEN
       #Quotient := #CounterTemp / 1;
       #CounterTemp := #CounterTemp MOD 1;
   ELSIF #TypeLayer = 2 THEN
       #Quotient := #CounterTemp / 2;
       #CounterTemp := #CounterTemp MOD 2;
   END_IF;

   IF #Quotient<>0 THEN
       "DB_Machine".CounterMachineInShift += #Quotient;
       "DB_Machine".CounterRaw += #Quotient;
   END_IF;
END_FUNCTION

FUNCTION "CheckSwitchPage" : Void   // FC20, SCL
{ S7_Optimized_Access := 'TRUE' }
VERSION : 0.1
   VAR_INPUT
      MaxPage : UDInt;
   END_VAR
   VAR_IN_OUT
      Action : UInt;   // 1: Tăng, 2: Giảm, 3 PLC reset
      PageCurrent : UDInt;
      EventChangePage : Bool;
   END_VAR
BEGIN
   IF #Action = 1 THEN
       IF #PageCurrent < #MaxPage THEN
           #PageCurrent += 1;
           #EventChangePage := TRUE;
       END_IF;
       #Action := 3;
   ELSIF #Action = 2 THEN
       IF #PageCurrent > 1 THEN
           #PageCurrent -= 1;
           #EventChangePage := TRUE;
       END_IF;
       #Action := 3;
   END_IF;
END_FUNCTION

FUNCTION "SortBufferLossInShift" : Void   // FC21, SCL
{ S7_Optimized_Access := 'TRUE' }
VERSION : 0.1
   VAR_INPUT
      page_current : UDInt;
   END_VAR
   VAR_IN_OUT
      number_data_in_shift : UDInt;
   END_VAR
   VAR_TEMP
      i : UInt;
      j : UInt;
      index : UDInt;
      IndexStart : USInt;
      IndexForGetDataShowHMI : USInt;
      total_data : UDInt;
      index_loss_group : UInt;
      index_loss_reason : UInt;
      index_bufer_src : UInt;
   END_VAR
BEGIN
   //"ClearBufferTempLossInShift"();

   //Gán buffer tạm
   FOR #i := 1 TO 100 DO
       "DB_Machine".buffer_index_sort[#i].id := "BuffersLoss_DB".buffer_loss_in_shift[#i].id;
       "DB_Machine".buffer_index_sort[#i].index_buffer := #i;
   END_FOR;


   //Sort giảm dần
   FOR #i := 1 TO 98 DO
       FOR #j := 1 TO 98 DO
           IF "DB_Machine".buffer_index_sort[#j].id < "DB_Machine".buffer_index_sort[#j + 1].id THEN
               "DB_Machine".value_temp := "DB_Machine".buffer_index_sort[#j];
               "DB_Machine".buffer_index_sort[#j] := "DB_Machine".buffer_index_sort[#j + 1];
               "DB_Machine".buffer_index_sort[#j + 1] := "DB_Machine".value_temp;
           END_IF;
       END_FOR;
   END_FOR;

   // Map lại dữ liệu HMI
   IF #number_data_in_shift > 0 THEN
       IF #page_current >= 1 AND #page_current <= 20 THEN
           FOR #IndexForGetDataShowHMI := 1 TO 5 DO
               // IF "DB_Machine".MachineStatus=2 OR "DB_Machine".MachineStatus=3 THEN
               //     // Statement section IF
               //     ;
               // ELSE

               // END_IF;




               // //Xử lý loss đang xảy ra do Server ko handle dc
               // IF #IndexForGetDataShowHMI=1 THEN
               //     // Statement section IF
               //     ;
               // ELSE

               // END_IF;




               #index := #IndexForGetDataShowHMI + (#page_current - 1) * 5;
               #index_bufer_src := "DB_Machine".buffer_index_sort[#index].index_buffer;

               IF #index_bufer_src >= 1 AND #index_bufer_src <= 100 THEN
                   IF "BuffersLoss_DB".buffer_loss_in_shift[#index].id > 0 THEN
                       "DB_DataHMI".DataLossInShiftShowHmiDTO[#IndexForGetDataShowHMI]."no." := UDINT_TO_UINT(#index);
                       "DB_DataHMI".DataLossInShiftShowHmiDTO[#IndexForGetDataShowHMI].id := "BuffersLoss_DB".buffer_loss_in_shift[#index_bufer_src].id;
                       "DB_DataHMI".DataLossInShiftShowHmiDTO[#IndexForGetDataShowHMI].LossCode := "BuffersLoss_DB".buffer_loss_in_shift[#index_bufer_src].losscode;

                       "DTL_to_DateString"("DTL" := "BuffersLoss_DB".buffer_loss_in_shift[#index_bufer_src].startTime,
                                           DateTimeString => "DB_DataHMI".DataLossInShiftShowHmiDTO[#IndexForGetDataShowHMI].StartDateAsStr);
                       "DTL_to_TimeString"("DTL" := "BuffersLoss_DB".buffer_loss_in_shift[#index_bufer_src].startTime,
                                           DateTimeString => "DB_DataHMI".DataLossInShiftShowHmiDTO[#IndexForGetDataShowHMI].StartTimeAsStr);

                       "DTL_to_DateString"("DTL" := "BuffersLoss_DB".buffer_loss_in_shift[#index_bufer_src].endTime,
                                           DateTimeString => "DB_DataHMI".DataLossInShiftShowHmiDTO[#IndexForGetDataShowHMI].EndDateAsStr);
                       "DTL_to_TimeString"("DTL" := "BuffersLoss_DB".buffer_loss_in_shift[#index_bufer_src].endTime,
                                           DateTimeString => "DB_DataHMI".DataLossInShiftShowHmiDTO[#IndexForGetDataShowHMI].EndTimeAsStr);

                       "Cvt_Duration_to_String"("Time(ms)" := "BuffersLoss_DB".buffer_loss_in_shift[#index_bufer_src].duration,
                                                ConvertTimeToStr => "DB_DataHMI".DataLossInShiftShowHmiDTO[#IndexForGetDataShowHMI].DurationAsStr);

                       #index_loss_reason := "BuffersLoss_DB".buffer_loss_in_shift[#index_bufer_src].losscode;
                       IF #index_loss_reason >= 1 AND #index_loss_reason <= 100 THEN
                           "DB_DataHMI".DataLossInShiftShowHmiDTO[#IndexForGetDataShowHMI].Description := "SettingsDB_LossDescription".loss_descriptions[#index_loss_reason].description;
                           #index_loss_group := "SettingsDB_LossDescription".loss_descriptions[#index_loss_reason].group_id;
                           IF #index_loss_group >= 1 AND #index_loss_group <= 10 THEN
                               "DB_DataHMI".DataLossInShiftShowHmiDTO[#IndexForGetDataShowHMI].GroupLossReason := "SettingsDB_LossDescription".loss_name_group[#index_loss_group];
                           END_IF;
                       END_IF;
                       "DB_DataHMI".DataLossInShiftShowHmiDTO[#IndexForGetDataShowHMI].IsHaveData := TRUE;
                   ELSE
                       "DB_DataHMI".DataLossInShiftShowHmiDTO[#IndexForGetDataShowHMI].IsHaveData := FALSE;
                   END_IF;

               END_IF;
           END_FOR;
       END_IF;
   END_IF;



















   // //"ClearBufferTempLossInShift"();

   // //Gán buffer tạm
   // FOR #i := 1 TO 100 DO
   //     "DB_Machine".buffer_index_sort[#i].id := "BuffersLoss_DB".buffer_loss_in_shift[#i].id;
   //     "DB_Machine".buffer_index_sort[#i].index_buffer := #i;
   // END_FOR;


   // //Sort giảm dần
   // FOR #i := 1 TO 98 DO
   //     FOR #j := 1 TO 98 DO
   //         IF "DB_Machine".buffer_index_sort[#j].id < "DB_Machine".buffer_index_sort[#j + 1].id THEN
   //             "DB_Machine".value_temp := "DB_Machine".buffer_index_sort[#j];
   //             "DB_Machine".buffer_index_sort[#j] := "DB_Machine".buffer_index_sort[#j + 1];
   //             "DB_Machine".buffer_index_sort[#j + 1] := "DB_Machine".value_temp;
   //         END_IF;
   //     END_FOR;
   // END_FOR;


   // //Clear buffer data show HMI
   // //"ClearTableShowHMI"("1: table in shift, 2:table historical, 3: table spare part":=1);

   // // Map lại dữ liệu HMI
   // IF #number_data_in_shift>0 THEN
   //     IF #page_current >= 1 AND #page_current <= 10 THEN
   //         FOR #IndexForGetDataShowHMI := 1 TO 5 DO
   //             #index := #IndexForGetDataShowHMI + (#page_current - 1) * 5;
   //             #index_bufer_src := "DB_Machine".buffer_index_sort[#index].index_buffer;

   //             IF #index_bufer_src>=1 AND #index_bufer_src<=100 THEN
   //                 IF "BuffersLoss_DB".buffer_loss_in_shift[#index].id > 0 THEN
   //                     "DB_DataHMI".DataLossInShiftShowHmiDTO[#IndexForGetDataShowHMI]."no." := UDINT_TO_UINT(#index);
   //                     "DB_DataHMI".DataLossInShiftShowHmiDTO[#IndexForGetDataShowHMI].id := "BuffersLoss_DB".buffer_loss_in_shift[#index_bufer_src].id;
   //                     "DB_DataHMI".DataLossInShiftShowHmiDTO[#IndexForGetDataShowHMI].LossCode := "BuffersLoss_DB".buffer_loss_in_shift[#index_bufer_src].losscode;

   //                     "DTL_to_DateString"("DTL" := "BuffersLoss_DB".buffer_loss_in_shift[#index_bufer_src].startTime,
   //                                         DateTimeString => "DB_DataHMI".DataLossInShiftShowHmiDTO[#IndexForGetDataShowHMI].StartDateAsStr);
   //                     "DTL_to_TimeString"("DTL" := "BuffersLoss_DB".buffer_loss_in_shift[#index_bufer_src].startTime,
   //                                         DateTimeString => "DB_DataHMI".DataLossInShiftShowHmiDTO[#IndexForGetDataShowHMI].StartTimeAsStr);

   //                     "DTL_to_DateString"("DTL" :="BuffersLoss_DB".buffer_loss_in_shift[#index_bufer_src].endTime,
   //                                         DateTimeString => "DB_DataHMI".DataLossInShiftShowHmiDTO[#IndexForGetDataShowHMI].EndDateAsStr);
   //                     "DTL_to_TimeString"("DTL" := "BuffersLoss_DB".buffer_loss_in_shift[#index_bufer_src].endTime,
   //                                         DateTimeString => "DB_DataHMI".DataLossInShiftShowHmiDTO[#IndexForGetDataShowHMI].EndTimeAsStr);

   //                     "Cvt_Duration_to_String"("Time(ms)" := "BuffersLoss_DB".buffer_loss_in_shift[#index_bufer_src].duration,
   //                                              ConvertTimeToStr => "DB_DataHMI".DataLossInShiftShowHmiDTO[#IndexForGetDataShowHMI].DurationAsStr);

   //                     #index_loss_reason :="BuffersLoss_DB".buffer_loss_in_shift[#index_bufer_src].losscode;
   //                     IF #index_loss_reason >= 1 AND #index_loss_reason <= 100 THEN
   //                         "DB_DataHMI".DataLossInShiftShowHmiDTO[#IndexForGetDataShowHMI].Description := "SettingsDB_LossDescription".loss_descriptions[#index_loss_reason].description;
   //                         #index_loss_group := "SettingsDB_LossDescription".loss_descriptions[#index_loss_reason].group_id;
   //                         IF #index_loss_group >= 1 AND #index_loss_group <= 10 THEN
   //                             "DB_DataHMI".DataLossInShiftShowHmiDTO[#IndexForGetDataShowHMI].GroupLossReason := "SettingsDB_LossDescription".loss_name_group[#index_loss_group];
   //                         END_IF;
   //                     END_IF;
   //                     "DB_DataHMI".DataLossInShiftShowHmiDTO[#IndexForGetDataShowHMI].IsHaveData := TRUE;
   //                 ELSE
   //                     "DB_DataHMI".DataLossInShiftShowHmiDTO[#IndexForGetDataShowHMI].IsHaveData := FALSE;
   //                 END_IF;

   //             END_IF;
   //         END_FOR;
   //     END_IF;
   // END_IF;
END_FUNCTION

FUNCTION "ReturnMaxPageFromTotalDataLossReason" : Void   // FC25, SCL
{ S7_Optimized_Access := 'TRUE' }
VERSION : 0.1
   VAR_INPUT
      DataPerPage : UInt;
      NumberData : UDInt;
      GroupId : UDInt;
   END_VAR
   VAR_OUTPUT
      TotalPage : UDInt;
   END_VAR
   VAR_TEMP
      Cnt : UInt;
      IndexFor : USInt;
      NumberDataTemp : UDInt;
   END_VAR
BEGIN
   IF #GroupId > 0 AND #GroupId <= 10 THEN
       #NumberDataTemp := 0;
       FOR #IndexFor := 1 TO 100 DO
           IF "SettingsDB_LossDescription".loss_descriptions[#IndexFor].group_id = #GroupId THEN
               #NumberDataTemp += 1;
           END_IF;
       END_FOR;
   ELSIF #GroupId = 0 THEN
       #NumberDataTemp := #NumberData;
   END_IF;


   IF #DataPerPage > 0 THEN
       #TotalPage := (#NumberDataTemp + #DataPerPage - 1) / #DataPerPage;
   ELSE
       #TotalPage := 0;
   END_IF;
END_FUNCTION

FUNCTION "LogStatusDb" : Void   // FC29, SCL
{ S7_Optimized_Access := 'TRUE' }
VERSION : 0.1
   VAR_INPUT
      status_machine : UInt;   // 1: Running, 2: Stop, 3: Idle, NG
   END_VAR
   VAR_IN_OUT
      index : USInt;
   END_VAR
BEGIN
   IF #index>="StatusMachineSendServerDB".min_index_buffer AND #index<="StatusMachineSendServerDB".max_index_buffer  THEN
       "StatusMachineSendServerDB".StatusMachineBuffer[#index].status := UINT_TO_USINT(#status_machine);
       "StatusMachineSendServerDB".StatusMachineBuffer[#index].time_start := "GlobalDB_RTC".RTC_Local;
       "StatusMachineSendServerDB".StatusMachineBuffer[#index].timer_end := "GlobalDB_RTC".RTC_Defaul;

       IF #index="StatusMachineSendServerDB".min_index_buffer THEN
           "StatusMachineSendServerDB".StatusMachineBuffer["StatusMachineSendServerDB".max_index_buffer].timer_end := "GlobalDB_RTC".RTC_Local;
       ELSE
           "StatusMachineSendServerDB".StatusMachineBuffer[#index-1].timer_end := "GlobalDB_RTC".RTC_Local;
       END_IF;

       #index += 1;
       IF #index>"StatusMachineSendServerDB".max_index_buffer THEN
           #index := 1;
       END_IF;

       "DB_Server".RequestServerUpdateBufferStatusMachine := 1;
   END_IF;

   "GLobalDB_LossManagementDB"."duration_status_curent(ms)" := 0;
END_FUNCTION

FUNCTION "QueryLossGroupFromLossReason" : Void   // FC30, SCL
{ S7_Optimized_Access := 'TRUE' }
VERSION : 0.1
   VAR_INPUT
      group_id : UInt;
      tab_index : UDInt;
   END_VAR
   VAR_TEMP
      index_for : UInt;
      data_temp : Array[1..100] of "ReasonLossHmi";
      index : USInt;
   END_VAR
BEGIN
   #index := 1;
   IF #group_id>=1 AND #group_id<=10 THEN
       FOR #index_for := 1 TO 100 DO
           IF "SettingsDB_LossDescription".loss_descriptions[#index_for].group_id = #group_id THEN
               #data_temp[#index].group_id := "SettingsDB_LossDescription".loss_descriptions[#index_for].group_id;
               #data_temp[#index].description := "SettingsDB_LossDescription".loss_descriptions[#index_for].description;
               #data_temp[#index].index_buffer := #index_for;
               #index += 1;
           END_IF;
       END_FOR;

       IF #tab_index >= 1 AND #tab_index <= 10 THEN
           FOR #index_for := 1 TO 10 DO
               IF #data_temp[#index_for + (#tab_index - 1) * 10].description = '' THEN
                   "DB_DataHMI".VisibleCheckboxLossReason[#index_for] := FALSE;
               ELSE
                   "DB_DataHMI".VisibleCheckboxLossReason[#index_for] := TRUE;
               END_IF;

               "DB_DataHMI".LossDescriptionHmiDTO[#index_for] := #data_temp[#index_for + (#tab_index - 1) * 10];
           END_FOR;
       END_IF;
   ELSIF #group_id=0 THEN
       FOR #index_for := 1 TO 100 DO
           #data_temp[#index].group_id := "SettingsDB_LossDescription".loss_descriptions[#index_for].group_id;
           #data_temp[#index].description := "SettingsDB_LossDescription".loss_descriptions[#index_for].description;
           #data_temp[#index].index_buffer := #index_for;
           #index += 1;
       END_FOR;

       IF #tab_index >= 1 AND #tab_index <= 10 THEN
           FOR #index_for := 1 TO 10 DO
               IF #data_temp[#index_for + (#tab_index - 1) * 10].description='' THEN
                   "DB_DataHMI".VisibleCheckboxLossReason[#index_for] := FALSE;
               ELSE
                   "DB_DataHMI".VisibleCheckboxLossReason[#index_for] := TRUE;
               END_IF;

               "DB_DataHMI".LossDescriptionHmiDTO[#index_for] := #data_temp[#index_for + (#tab_index - 1) * 10];
           END_FOR;
       END_IF;
   END_IF;
END_FUNCTION

FUNCTION "CheckCheckBoxAssign" : Void   // FC31, SCL
{ S7_Optimized_Access := 'TRUE' }
VERSION : 0.1
   VAR_INPUT
      index_checkbox : UInt;   // 0: không chọn, còn lại tương ứng từ 1->10
   END_VAR
   VAR_IN_OUT
      array_check_box : Array[1..10] of UInt;
   END_VAR
   VAR_TEMP
      index_for : USInt;
   END_VAR
BEGIN
   FOR #index_for := 1 TO 10 DO
       IF #index_checkbox >= 1 AND #index_checkbox <= 10 THEN
           IF #index_for=#index_checkbox THEN 
               #array_check_box[#index_for] := 1;
           ELSE
               #array_check_box[#index_for] := 0;
           END_IF;
       ELSE
           #array_check_box[#index_for] := 0;
       END_IF;
   END_FOR;
END_FUNCTION

FUNCTION "ShowDataLossGroup_Reason" : Void   // FC32, SCL
{ S7_Optimized_Access := 'TRUE' }
VERSION : 0.1
   VAR_INPUT
      tab_index : UDInt;
      "1: LossGroup, 2: LossReason" : USInt;   // 1: LossGroup, 2: LossReason, NG
   END_VAR
   VAR_TEMP
      index : UDInt;
      index_for : USInt;
   END_VAR
BEGIN
   IF #"1: LossGroup, 2: LossReason"=1 THEN
       IF #tab_index >= 1 THEN
           FOR #index_for := 1 TO 10 DO
               #index := (#tab_index - 1) * 10 + #index_for;
               IF #index <= 100 THEN
                   "DB_DataHMI".LossDescriptionHmiDTO[#index_for].group_id := "SettingsDB_LossDescription".loss_descriptions[#index].group_id;
                   "DB_DataHMI".LossDescriptionHmiDTO[#index_for].description := "SettingsDB_LossDescription".loss_descriptions[#index].description;
               END_IF;
           END_FOR;
       END_IF;
   ELSIF #"1: LossGroup, 2: LossReason"=2 THEN
       IF #tab_index >= 1 THEN
           FOR #index_for := 1 TO 10 DO
               #index := (#tab_index - 1) * 10 + #index_for;
               IF #index <= 100 THEN
                   "DB_DataHMI".LossDescriptionHmiDTO[#index_for].group_id := "SettingsDB_LossDescription".loss_descriptions[#index].group_id;
                   "DB_DataHMI".LossDescriptionHmiDTO[#index_for].description := "SettingsDB_LossDescription".loss_descriptions[#index].description;
               END_IF;
           END_FOR;
       END_IF;
   END_IF;
END_FUNCTION

FUNCTION "ReturnPageFromTotalData" : Void   // FC40, SCL
{ S7_Optimized_Access := 'TRUE' }
VERSION : 0.1
   VAR_INPUT
      total_data : UDInt;
      data_per_page : UInt;
   END_VAR
   VAR_OUTPUT
      total_page : UDInt;
   END_VAR
BEGIN
   IF #total_data=0 THEN
       #total_page := 1;
   ELSE
       IF #data_per_page > 0 THEN
           #total_page := (#total_data + #data_per_page - 1) / #data_per_page;
       ELSE
           #total_page := 1;
       END_IF;
   END_IF;
END_FUNCTION

ORGANIZATION_BLOCK "Main"   // OB1, LAD, ProgramCycle
TITLE = "Main Program Sweep (Cycle)"
{ S7_Optimized_Access := 'TRUE' }
VERSION : 0.1
// Write by:
   VAR_INPUT
      Initial_Call : Bool;   // Initial call of this OB
      Remanence : Bool;   // =True, if remanent data are available
   END_VAR
   VAR_TEMP
      tempC : DInt;
      scale_real_tmp : Real;
      Real_Temperature : Real;
      Real_Current : Real;
      "Real_Pressure IN" : Real;
      "Real_Pressure Out" : Real;
      Speed : DInt;
      SpeedMotor : DInt;
      b_tmp : Bool;
      Year : UInt;
      Month : UInt;
      Day : UInt;
      Hour : UInt;
      Minute : UInt;
      Second : UInt;
      bMachineRun : Bool;
      Dint_Temperature : DInt;
      Dint_Current : DInt;
      Dint_PressureIN : DInt;
      Dint_PressureOut : DInt;
      total_run_time : Time;
      total_stop_time : Time;
      tmpIsDiff : Bool;
      tmp_tartTimeAsStr : String;
      total_page : USInt;
      max_slotId : Int;
      min_slotId : Int;
      SignalRaisingCnt : Bool;
      loss_group_id_temp : UInt;
      index_for : UInt;
      id_test : UDInt;
      bit_search_spare_part : Bool;
      event_chage_page_loss_description : Bool;
      event_chage_page_loss_in_shift : Bool;
      event_chage_page_loss_historical : Bool;
      pulse_check_connect_hmi : Bool;
      event_chage_page_spare_part : Bool;
      signal_relay_speed : Bool;
   END_VAR
   VAR_TEMP   // added for the SCL form of the ladder/FBD networks
      _w1 : Bool;
      _w2 : Bool;
      _w3 : Bool;
      _w4 : Bool;
      _w5 : Bool;
      _w6 : Bool;
   END_VAR
BEGIN

REGION Network 1: MQTT
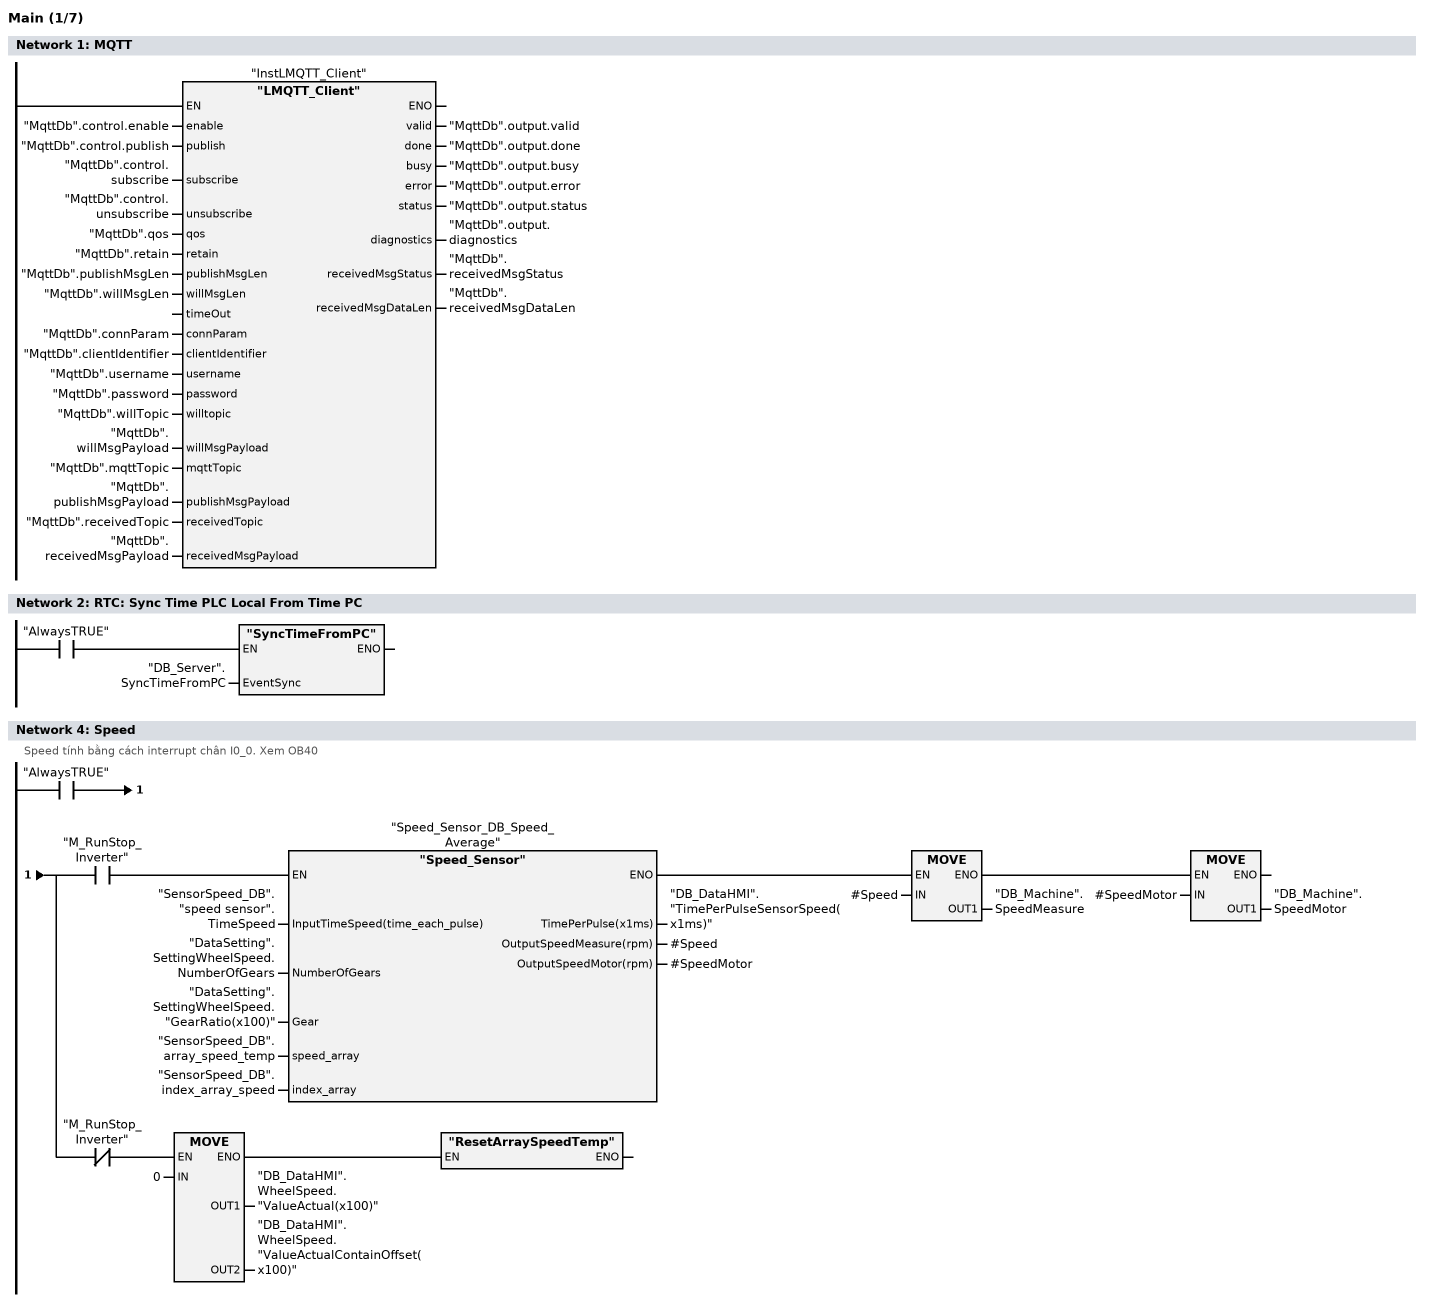
   RUNG wire#powerrail
      "InstLMQTT_Client"(enable := "MqttDb".control.enable, publish := "MqttDb".control.publish, subscribe := "MqttDb".control.subscribe, unsubscribe := "MqttDb".control.unsubscribe, qos := "MqttDb".qos, retain := "MqttDb".retain, publishMsgLen := "MqttDb".publishMsgLen, willMsgLen := "MqttDb".willMsgLen, timeOut :=, connParam := "MqttDb".connParam, clientIdentifier := "MqttDb".clientIdentifier, username := "MqttDb".username, password := "MqttDb".password, willtopic := "MqttDb".willTopic, willMsgPayload := "MqttDb".willMsgPayload, mqttTopic := "MqttDb".mqttTopic, publishMsgPayload := "MqttDb".publishMsgPayload, receivedTopic := "MqttDb".receivedTopic, receivedMsgPayload := "MqttDb".receivedMsgPayload, valid => "MqttDb".output.valid, done => "MqttDb".output.done, busy => "MqttDb".output.busy, error => "MqttDb".output.error, status => "MqttDb".output.status, diagnostics => "MqttDb".output.diagnostics, receivedMsgStatus => "MqttDb".receivedMsgStatus, receivedMsgDataLen => "MqttDb".receivedMsgDataLen)
   END_RUNG
   // the same network as SCL:
   "InstLMQTT_Client"(enable := "MqttDb".control.enable,   // "LMQTT_Client"
                      publish := "MqttDb".control.publish,
                      subscribe := "MqttDb".control.subscribe,
                      unsubscribe := "MqttDb".control.unsubscribe,
                      qos := "MqttDb".qos,
                      retain := "MqttDb".retain,
                      publishMsgLen := "MqttDb".publishMsgLen,
                      willMsgLen := "MqttDb".willMsgLen,
                      connParam := "MqttDb".connParam,
                      clientIdentifier := "MqttDb".clientIdentifier,
                      username := "MqttDb".username,
                      password := "MqttDb".password,
                      willtopic := "MqttDb".willTopic,
                      willMsgPayload := "MqttDb".willMsgPayload,
                      mqttTopic := "MqttDb".mqttTopic,
                      publishMsgPayload := "MqttDb".publishMsgPayload,
                      receivedTopic := "MqttDb".receivedTopic,
                      receivedMsgPayload := "MqttDb".receivedMsgPayload,
                      valid => "MqttDb".output.valid,
                      done => "MqttDb".output.done,
                      busy => "MqttDb".output.busy,
                      error => "MqttDb".output.error,
                      status => "MqttDb".output.status,
                      diagnostics => "MqttDb".output.diagnostics,
                      receivedMsgStatus => "MqttDb".receivedMsgStatus,
                      receivedMsgDataLen => "MqttDb".receivedMsgDataLen);
END_REGION

REGION Network 2: RTC: Sync Time PLC Local From Time PC
   RUNG wire#powerrail
      Contact( "AlwaysTRUE" )
      "SyncTimeFromPC"(EventSync := "DB_Server".SyncTimeFromPC)
   END_RUNG
   // the same network as SCL:
   IF "AlwaysTRUE" THEN "SyncTimeFromPC"(EventSync := "DB_Server".SyncTimeFromPC); END_IF;
END_REGION

REGION Network 3 (SCL): Mapping input & analog
   "TagTest".TimeLastOnPlcRealTime := "GlobalDB_RTC".RTC_Local;
   "DB_DataHMI".Year_HMI:= UINT_TO_INT( "GlobalDB_RTC".RTC_Local.YEAR);
   "DB_DataHMI".Month_HMI := USINT_TO_INT("GlobalDB_RTC".RTC_Local.MONTH);
   "DB_DataHMI".Day_HMI := USINT_TO_INT("GlobalDB_RTC".RTC_Local.DAY);
   "DB_DataHMI".Hour_HMI := USINT_TO_INT("GlobalDB_RTC".RTC_Local.HOUR);
   "DB_DataHMI".Minute_HMI := USINT_TO_INT("GlobalDB_RTC".RTC_Local.MINUTE);
   "DB_DataHMI".Second_HMI := USINT_TO_INT("GlobalDB_RTC".RTC_Local.SECOND);

   IF "GLobalDB_LossManagementDB".index_buffer_loss_in_shift_current=0 THEN
       "GLobalDB_LossManagementDB".index_buffer_loss_in_shift_current := 1;
   END_IF;


   //Bộ giải mã
   "DB_Machine".AnalogSensorMin := 0;
   "DB_Machine".AnalogSensorMax := 27648;

   "DB_DataHMI".AnalogSensorMin := 0;
   "DB_DataHMI".AnalogSensorMax := 27648;

   //Mapping Analog 
   // "M_Current" := "AI1_Current";
   // "M_Analog_Spare" := "AI2_Spare";
   // "M_Temperature" := "AI3_Temperature";
   // "M_Pressure Out" := "AI4_Pressure_Out";

   // IF "TagTest".RandomAnalog THEN
   //     "M_Temperature" := "RandomAnalogs".Temp_Analog;
   //     "M_Current" := "RandomAnalogs".Current_Analog;
   //     "M_Analog_Spare" := "RandomAnalogs".Pressure_Analog;
   //     "M_Pressure Out" := "RandomAnalogs".Pressure_Analog;
   // ELSE
   //     // "M_Current" := "AI_Module_Ch00_Pressure_In";
   //     // "M_Analog_Spare" := "AI_Module_Ch01__Pressure_Out";
   //     // "M_Temperature" := "AI_Module_Ch02_Temperature";
   //     // "M_Pressure Out" := "AI_Module_Ch03";
   //     // 
   //     "M_Current" := "AI_PLC_Ch00_Current";

   //     "M_Pressure Out" := "AI_Module_Ch01__Pressure_Out";
   //     "M_Temperature" := "AI_Module_Ch02_Temperature";
   //     "M_Analog_Spare" := "AI_Module_Ch03";
   // END_IF;
   // 

   "M_Current" := "AI_PLC_Ch00_Current";
   "M_AnalogPlc_Spare" := "AI_PLC_Ch01";

   "M_Pressure In" := "AI_Module_Ch01__Pressure_Out";
   "M_Pressure Out" := "AI_Module_Ch00_Pressure_In";
   "M_Temperature" := "AI_Module_Ch02_Temperature";
   "M_AnalogModule_Spare" := "AI_Module_Ch03";

   //Mapping IO
   "M_Speed" := "I0_0_Speed";
   "M_RunStop_Machine" := "I0_1_RunStop_Machine";
   "M_Xilanh_Push" := "I0_2_Signal_Xilanh_Push";
   "M_Pedal" := "I0_3_Signal_Pedal";
   "M_RunStop_Inverter" := "I0_4_RunStop_Inverter";

   "Input 5 Spare" := "I0_5_Spare";
   "Input 6 Spare" := "I0_6_Spare";
   "Input 7 Spare" := "I0_7_Spare";
END_REGION

REGION Network 4: Speed
   // Speed tính bằng cách interrupt chân I0_0. Xem OB40
   RUNG wire#powerrail
      Contact( "AlwaysTRUE" )
      wire#w1
      Contact( "M_RunStop_Inverter" )
      "Speed_Sensor_DB_Speed_Average"("InputTimeSpeed(time_each_pulse)" := "SensorSpeed_DB"."speed sensor".TimeSpeed, NumberOfGears := "DataSetting".SettingWheelSpeed.NumberOfGears, Gear := "DataSetting".SettingWheelSpeed."GearRatio(x100)", speed_array := "SensorSpeed_DB".array_speed_temp, index_array := "SensorSpeed_DB".index_array_speed, "TimePerPulse(x1ms)" => "DB_DataHMI"."TimePerPulseSensorSpeed(x1ms)", "OutputSpeedMeasure(rpm)" => #Speed, "OutputSpeedMotor(rpm)" => #SpeedMotor)
      Move(in := #Speed, out1 => "DB_Machine".SpeedMeasure)
      Move(in := #SpeedMotor, out1 => "DB_Machine".SpeedMotor)
   END_RUNG
   RUNG wire#w1
      I_Contact( "M_RunStop_Inverter" )
      Move(in := 0, out1 => "DB_DataHMI".WheelSpeed."ValueActual(x100)", out2 => "DB_DataHMI".WheelSpeed."ValueActualContainOffset(x100)")
      "ResetArraySpeedTemp"()
   END_RUNG
   // the same network as SCL:
   #_w2 := "AlwaysTRUE";
   "Speed_Sensor_DB_Speed_Average"(EN := "AlwaysTRUE" AND "M_RunStop_Inverter",   // "Speed_Sensor"
                           "InputTimeSpeed(time_each_pulse)" := "SensorSpeed_DB"."speed sensor".TimeSpeed,
                           NumberOfGears := "DataSetting".SettingWheelSpeed.NumberOfGears,
                           Gear := "DataSetting".SettingWheelSpeed."GearRatio(x100)",
                           speed_array := "SensorSpeed_DB".array_speed_temp,
                           index_array := "SensorSpeed_DB".index_array_speed,
                           "TimePerPulse(x1ms)" => "DB_DataHMI"."TimePerPulseSensorSpeed(x1ms)",
                           "OutputSpeedMeasure(rpm)" => #Speed,
                           "OutputSpeedMotor(rpm)" => #SpeedMotor,
                           ENO => #_w1);
   IF #_w1 THEN
       "DB_Machine".SpeedMeasure := #Speed;
       "DB_Machine".SpeedMotor := #SpeedMotor;
   END_IF;
   IF #_w2 AND NOT "M_RunStop_Inverter" THEN
       "DB_DataHMI".WheelSpeed."ValueActual(x100)" := 0;
       "DB_DataHMI".WheelSpeed."ValueActualContainOffset(x100)" := 0;
       "ResetArraySpeedTemp"();
   END_IF;
END_REGION

REGION Network 5: Check tăng Counter
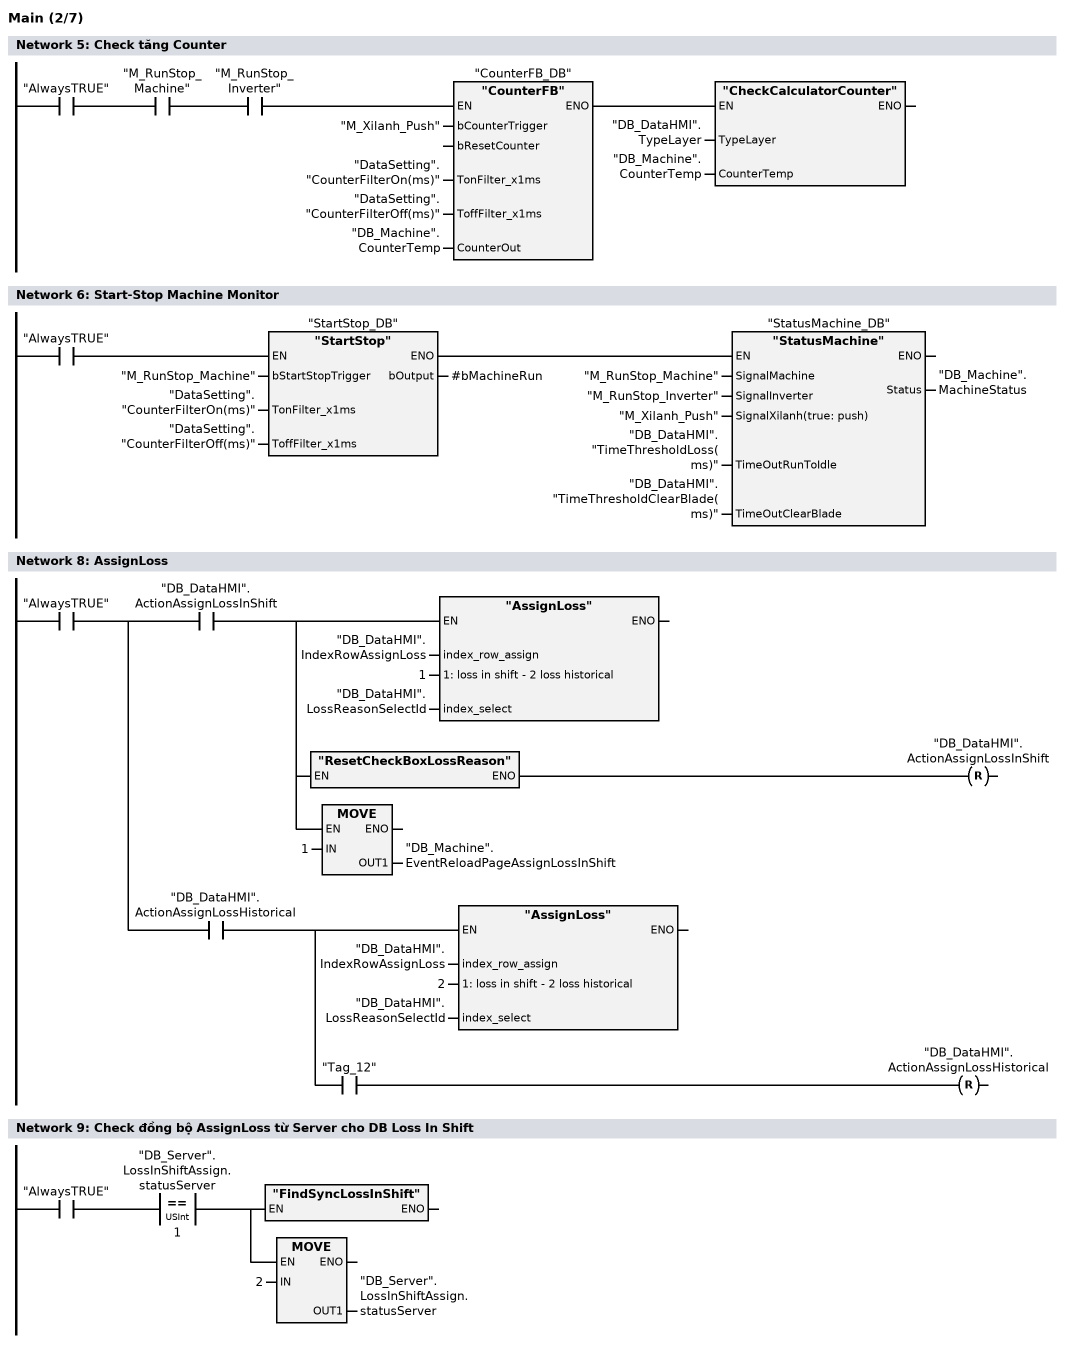
   RUNG wire#powerrail
      Contact( "AlwaysTRUE" )
      Contact( "M_RunStop_Machine" )
      Contact( "M_RunStop_Inverter" )
      "CounterFB_DB"(bCounterTrigger := "M_Xilanh_Push", bResetCounter :=, TonFilter_x1ms := "DataSetting"."CounterFilterOn(ms)", ToffFilter_x1ms := "DataSetting"."CounterFilterOff(ms)", CounterOut := "DB_Machine".CounterTemp)
      "CheckCalculatorCounter"(TypeLayer := "DB_DataHMI".TypeLayer, CounterTemp := "DB_Machine".CounterTemp)
   END_RUNG
   // the same network as SCL:
   "CounterFB_DB"(EN := "AlwaysTRUE" AND "M_RunStop_Machine" AND "M_RunStop_Inverter",   // "CounterFB"
                  bCounterTrigger := "M_Xilanh_Push",
                  TonFilter_x1ms := "DataSetting"."CounterFilterOn(ms)",
                  ToffFilter_x1ms := "DataSetting"."CounterFilterOff(ms)",
                  CounterOut := "DB_Machine".CounterTemp,
                  ENO => #_w1);
   IF #_w1 THEN
       "CheckCalculatorCounter"(TypeLayer := "DB_DataHMI".TypeLayer, CounterTemp := "DB_Machine".CounterTemp);
   END_IF;
END_REGION

REGION Network 6: Start-Stop Machine Monitor
   RUNG wire#powerrail
      Contact( "AlwaysTRUE" )
      "StartStop_DB"(bStartStopTrigger := "M_RunStop_Machine", TonFilter_x1ms := "DataSetting"."CounterFilterOn(ms)", ToffFilter_x1ms := "DataSetting"."CounterFilterOff(ms)", bOutput => #bMachineRun)
      "StatusMachine_DB"(SignalMachine := "M_RunStop_Machine", SignalInverter := "M_RunStop_Inverter", "SignalXilanh(true: push)" := "M_Xilanh_Push", TimeOutRunToIdle := "DB_DataHMI"."TimeThresholdLoss(ms)", TimeOutClearBlade := "DB_DataHMI"."TimeThresholdClearBlade(ms)", Status => "DB_Machine".MachineStatus)
   END_RUNG
   // the same network as SCL:
   "StartStop_DB"(EN := "AlwaysTRUE",   // "StartStop"
                  bStartStopTrigger := "M_RunStop_Machine",
                  TonFilter_x1ms := "DataSetting"."CounterFilterOn(ms)",
                  ToffFilter_x1ms := "DataSetting"."CounterFilterOff(ms)",
                  bOutput => #bMachineRun,
                  ENO => #_w1);
   IF #_w1 THEN
       "StatusMachine_DB"(SignalMachine := "M_RunStop_Machine",   // "StatusMachine"
                          SignalInverter := "M_RunStop_Inverter",
                          "SignalXilanh(true: push)" := "M_Xilanh_Push",
                          TimeOutRunToIdle := "DB_DataHMI"."TimeThresholdLoss(ms)",
                          TimeOutClearBlade := "DB_DataHMI"."TimeThresholdClearBlade(ms)",
                          Status => "DB_Machine".MachineStatus);
   END_IF;
END_REGION

REGION Network 7 (SCL): Log Loss nếu đổi trạng thái
   "CheckMoveDataLossCurrent"();

   IF "DB_Machine".MachineStatus <>"DB_Machine".MachineStatusPrevious THEN
       //DB Status To Server
       "LogStatusDb"(status_machine:="DB_Machine".MachineStatus,
                     index:="StatusMachineSendServerDB".index_current);
       IF "DB_Machine".MachineStatusPrevious = 2 OR "DB_Machine".MachineStatusPrevious = 3 THEN
           //Log Loss
           "LogLoss"(status := "DB_Machine".MachineStatusPrevious,
                     index_buffer := "GLobalDB_LossManagementDB".index_buffer_loss_in_shift_current);
           "ClearTableShowHMI"(1);
           // ELSIF "DB_Machine".MachineStatusPrevious=1 THEN
           //     "DB_Machine".NumberLossInShift += 1;
       END_IF;

       IF "DB_Machine".MachineStatusPrevious=1 AND "DB_Machine".MachineStatus=2  THEN
           "DB_Machine".NumberLossInShift += 1;
       ELSIF "DB_Machine".MachineStatusPrevious=1 AND "DB_Machine".MachineStatus=3  THEN
           "DB_Machine".NumberLossInShift += 1;
       ELSIF "DB_Machine".MachineStatusPrevious=2 AND "DB_Machine".MachineStatus=3  THEN
           "DB_Machine".NumberLossInShift += 1;
       ELSIF "DB_Machine".MachineStatusPrevious=3 AND "DB_Machine".MachineStatus=2  THEN
           "DB_Machine".NumberLossInShift += 1;
       END_IF;



       //Status Current
       "GLobalDB_LossManagementDB".current_status_machine.startTime := "GlobalDB_RTC".RTC_Local;

       //Event
       "DB_Machine".EventReloadPageAssignLossInShift := 1;
       "DB_Server".RequestServerUpdateLossInShift := 1;
       "DB_Machine".MachineStatusPrevious := "DB_Machine".MachineStatus;

       //Clear flag nếu qua loss mới
       "DB_DataHMI".FlagCancelAssignLossCurrent := FALSE;
   END_IF;
END_REGION

REGION Network 8: AssignLoss
   RUNG wire#powerrail
      Contact( "AlwaysTRUE" )
      wire#w1
      Contact( "DB_DataHMI".ActionAssignLossInShift )
      wire#w2
      "AssignLoss"(index_row_assign := "DB_DataHMI".IndexRowAssignLoss, "1: loss in shift - 2 loss historical" := 1, index_select := "DB_DataHMI".LossReasonSelectId)
   END_RUNG
   RUNG wire#w2
      "ResetCheckBoxLossReason"()
      R_Coil( "DB_DataHMI".ActionAssignLossInShift )
   END_RUNG
   RUNG wire#w2
      Move(in := 1, out1 => "DB_Machine".EventReloadPageAssignLossInShift)
   END_RUNG
   RUNG wire#w1
      Contact( "DB_DataHMI".ActionAssignLossHistorical )
      wire#w3
      "AssignLoss"(index_row_assign := "DB_DataHMI".IndexRowAssignLoss, "1: loss in shift - 2 loss historical" := 2, index_select := "DB_DataHMI".LossReasonSelectId)
   END_RUNG
   RUNG wire#w3
      Contact( "Tag_12" )
      R_Coil( "DB_DataHMI".ActionAssignLossHistorical )
   END_RUNG
   // the same network as SCL:
   #_w1 := "AlwaysTRUE";
   #_w2 := "AlwaysTRUE" AND "DB_DataHMI".ActionAssignLossInShift;
   IF #_w2 THEN
       "AssignLoss"(index_row_assign := "DB_DataHMI".IndexRowAssignLoss,
                    "1: loss in shift - 2 loss historical" := 1,
                    index_select := "DB_DataHMI".LossReasonSelectId);
   END_IF;
   "ResetCheckBoxLossReason"(EN := #_w2, ENO => #_w3);
   IF #_w3 THEN "DB_DataHMI".ActionAssignLossInShift := FALSE; END_IF;
   IF #_w2 THEN "DB_Machine".EventReloadPageAssignLossInShift := 1; END_IF;
   #_w4 := #_w1 AND "DB_DataHMI".ActionAssignLossHistorical;
   IF #_w4 THEN
       "AssignLoss"(index_row_assign := "DB_DataHMI".IndexRowAssignLoss,
                    "1: loss in shift - 2 loss historical" := 2,
                    index_select := "DB_DataHMI".LossReasonSelectId);
   END_IF;
   IF #_w4 AND "Tag_12" THEN "DB_DataHMI".ActionAssignLossHistorical := FALSE; END_IF;
END_REGION

REGION Network 9: Check đồng bộ AssignLoss từ Server cho DB Loss In Shift
   RUNG wire#powerrail
      Contact( "AlwaysTRUE" )
      { S7_Templates := "SrcType := USInt" } EQ_Contact(in1 := "DB_Server".LossInShiftAssign.statusServer, in2 := 1)
      wire#w1
      "FindSyncLossInShift"()
   END_RUNG
   RUNG wire#w1
      Move(in := 2, out1 => "DB_Server".LossInShiftAssign.statusServer)
   END_RUNG
   // the same network as SCL:
   #_w1 := "AlwaysTRUE" AND ("DB_Server".LossInShiftAssign.statusServer = 1);
   IF #_w1 THEN
       "FindSyncLossInShift"();
       "DB_Server".LossInShiftAssign.statusServer := 2;
   END_IF;
END_REGION

REGION Network 10: Tính số Page Kiểm tra chuyển Page
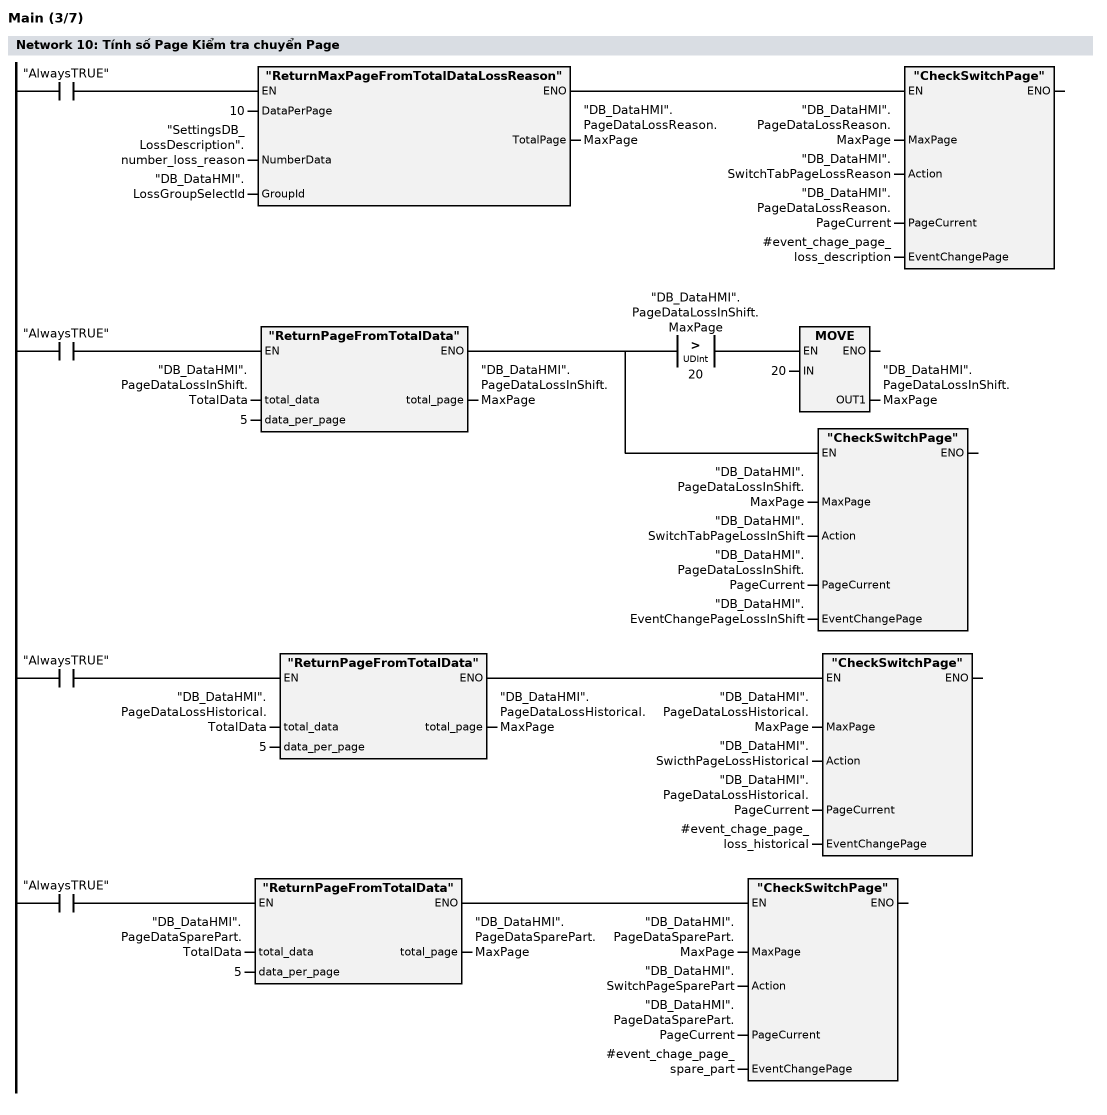
   RUNG wire#powerrail
      Contact( "AlwaysTRUE" )
      "ReturnMaxPageFromTotalDataLossReason"(DataPerPage := 10, NumberData := "SettingsDB_LossDescription".number_loss_reason, GroupId := "DB_DataHMI".LossGroupSelectId, TotalPage => "DB_DataHMI".PageDataLossReason.MaxPage)
      "CheckSwitchPage"(MaxPage := "DB_DataHMI".PageDataLossReason.MaxPage, Action := "DB_DataHMI".SwitchTabPageLossReason, PageCurrent := "DB_DataHMI".PageDataLossReason.PageCurrent, EventChangePage := #event_chage_page_loss_description)
   END_RUNG
   RUNG wire#powerrail
      Contact( "AlwaysTRUE" )
      "ReturnPageFromTotalData"(total_data := "DB_DataHMI".PageDataLossInShift.TotalData, data_per_page := 5, total_page => "DB_DataHMI".PageDataLossInShift.MaxPage)
      wire#w1
      { S7_Templates := "SrcType := UDInt" } GT_Contact(in1 := "DB_DataHMI".PageDataLossInShift.MaxPage, in2 := 20)
      Move(in := 20, out1 => "DB_DataHMI".PageDataLossInShift.MaxPage)
   END_RUNG
   RUNG wire#w1
      "CheckSwitchPage"(MaxPage := "DB_DataHMI".PageDataLossInShift.MaxPage, Action := "DB_DataHMI".SwitchTabPageLossInShift, PageCurrent := "DB_DataHMI".PageDataLossInShift.PageCurrent, EventChangePage := "DB_DataHMI".EventChangePageLossInShift)
   END_RUNG
   RUNG wire#powerrail
      Contact( "AlwaysTRUE" )
      "ReturnPageFromTotalData"(total_data := "DB_DataHMI".PageDataLossHistorical.TotalData, data_per_page := 5, total_page => "DB_DataHMI".PageDataLossHistorical.MaxPage)
      "CheckSwitchPage"(MaxPage := "DB_DataHMI".PageDataLossHistorical.MaxPage, Action := "DB_DataHMI".SwicthPageLossHistorical, PageCurrent := "DB_DataHMI".PageDataLossHistorical.PageCurrent, EventChangePage := #event_chage_page_loss_historical)
   END_RUNG
   RUNG wire#powerrail
      Contact( "AlwaysTRUE" )
      "ReturnPageFromTotalData"(total_data := "DB_DataHMI".PageDataSparePart.TotalData, data_per_page := 5, total_page => "DB_DataHMI".PageDataSparePart.MaxPage)
      "CheckSwitchPage"(MaxPage := "DB_DataHMI".PageDataSparePart.MaxPage, Action := "DB_DataHMI".SwitchPageSparePart, PageCurrent := "DB_DataHMI".PageDataSparePart.PageCurrent, EventChangePage := #event_chage_page_spare_part)
   END_RUNG
   // the same network as SCL:
   "ReturnMaxPageFromTotalDataLossReason"(EN := "AlwaysTRUE",
                           DataPerPage := 10,
                           NumberData := "SettingsDB_LossDescription".number_loss_reason,
                           GroupId := "DB_DataHMI".LossGroupSelectId,
                           TotalPage => "DB_DataHMI".PageDataLossReason.MaxPage,
                           ENO => #_w1);
   IF #_w1 THEN
       "CheckSwitchPage"(MaxPage := "DB_DataHMI".PageDataLossReason.MaxPage,
                         Action := "DB_DataHMI".SwitchTabPageLossReason,
                         PageCurrent := "DB_DataHMI".PageDataLossReason.PageCurrent,
                         EventChangePage := #event_chage_page_loss_description);
   END_IF;
   "ReturnPageFromTotalData"(EN := "AlwaysTRUE",
                           total_data := "DB_DataHMI".PageDataLossInShift.TotalData,
                           data_per_page := 5,
                           total_page => "DB_DataHMI".PageDataLossInShift.MaxPage,
                           ENO => #_w2);
   IF #_w2 AND ("DB_DataHMI".PageDataLossInShift.MaxPage > 20) THEN
       "DB_DataHMI".PageDataLossInShift.MaxPage := 20;
   END_IF;
   IF #_w2 THEN
       "CheckSwitchPage"(MaxPage := "DB_DataHMI".PageDataLossInShift.MaxPage,
                         Action := "DB_DataHMI".SwitchTabPageLossInShift,
                         PageCurrent := "DB_DataHMI".PageDataLossInShift.PageCurrent,
                         EventChangePage := "DB_DataHMI".EventChangePageLossInShift);
   END_IF;
   "ReturnPageFromTotalData"(EN := "AlwaysTRUE",
                           total_data := "DB_DataHMI".PageDataLossHistorical.TotalData,
                           data_per_page := 5,
                           total_page => "DB_DataHMI".PageDataLossHistorical.MaxPage,
                           ENO => #_w3);
   IF #_w3 THEN
       "CheckSwitchPage"(MaxPage := "DB_DataHMI".PageDataLossHistorical.MaxPage,
                         Action := "DB_DataHMI".SwicthPageLossHistorical,
                         PageCurrent := "DB_DataHMI".PageDataLossHistorical.PageCurrent,
                         EventChangePage := #event_chage_page_loss_historical);
   END_IF;
   "ReturnPageFromTotalData"(EN := "AlwaysTRUE",
                           total_data := "DB_DataHMI".PageDataSparePart.TotalData,
                           data_per_page := 5,
                           total_page => "DB_DataHMI".PageDataSparePart.MaxPage,
                           ENO => #_w4);
   IF #_w4 THEN
       "CheckSwitchPage"(MaxPage := "DB_DataHMI".PageDataSparePart.MaxPage,
                         Action := "DB_DataHMI".SwitchPageSparePart,
                         PageCurrent := "DB_DataHMI".PageDataSparePart.PageCurrent,
                         EventChangePage := #event_chage_page_spare_part);
   END_IF;
END_REGION

REGION Network 11: Show Loss Description Loss và NameGroup
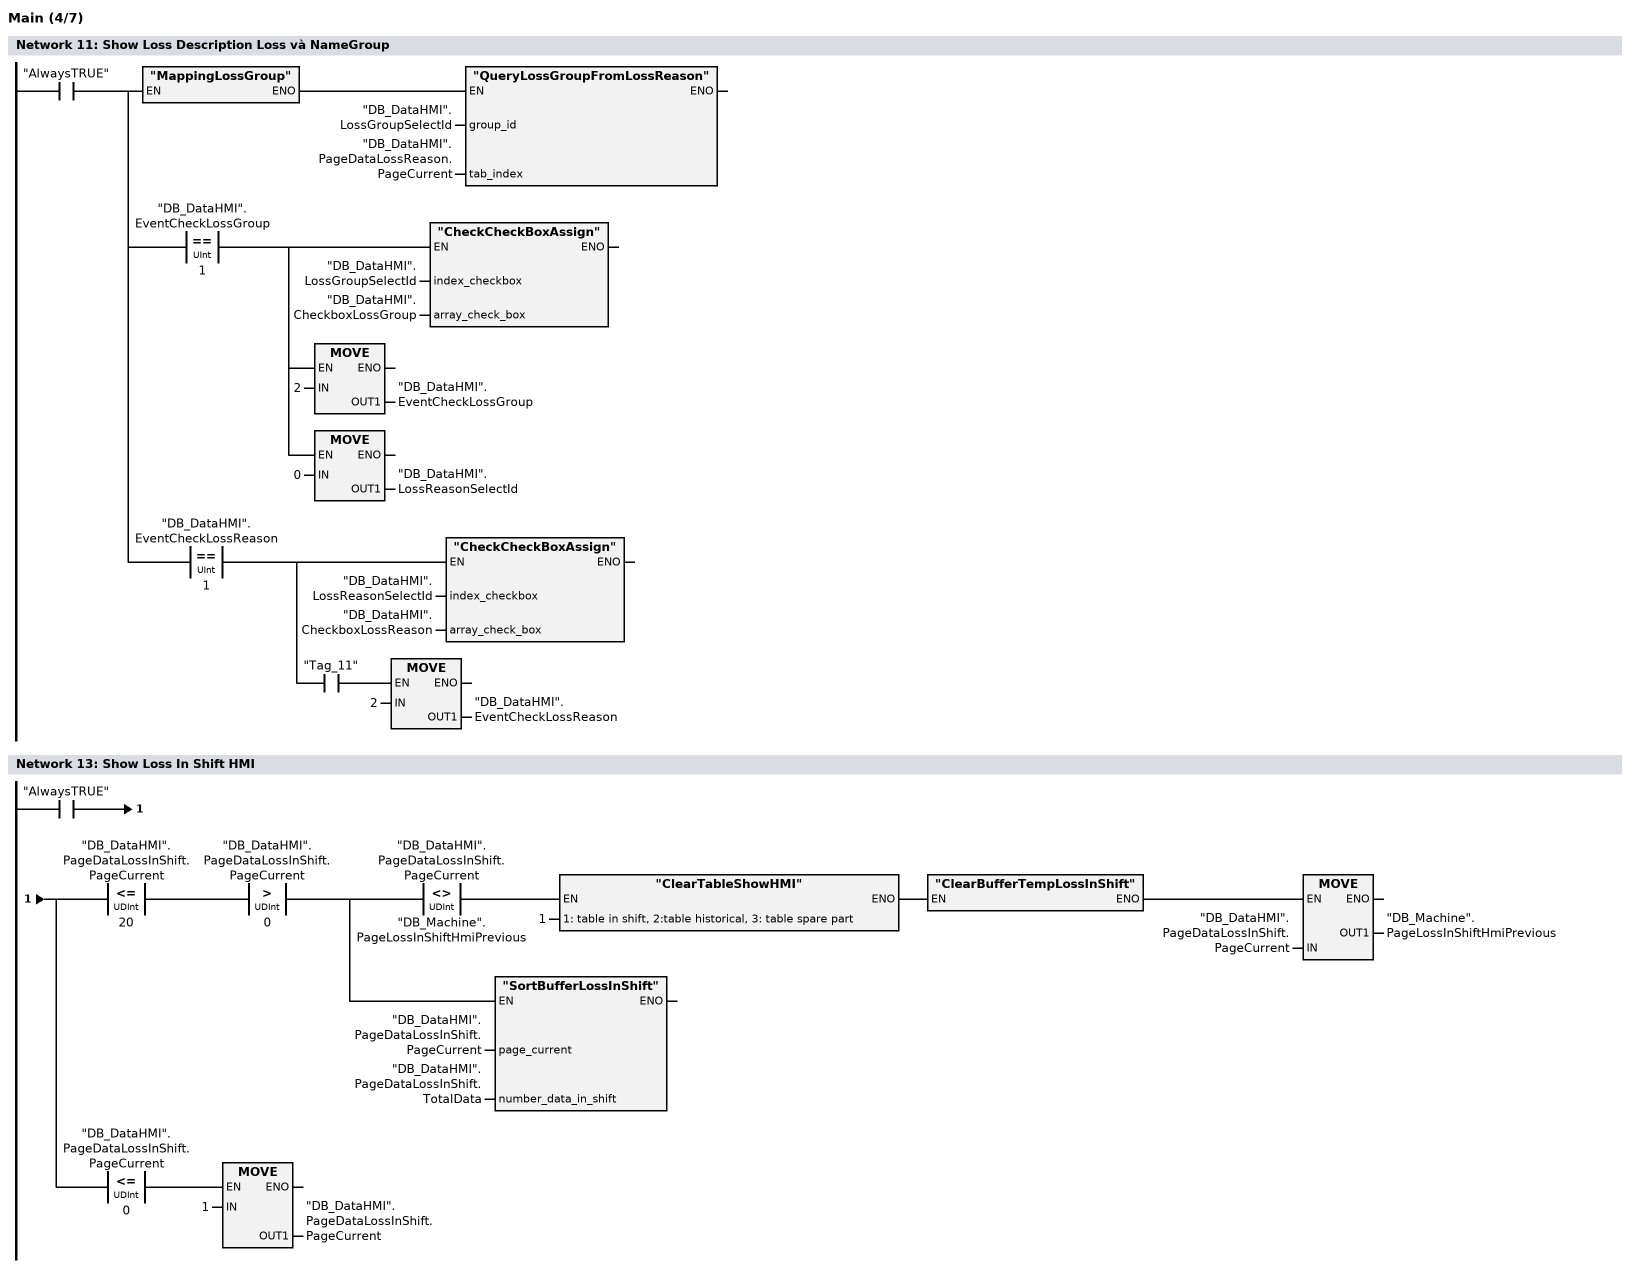
   RUNG wire#powerrail
      Contact( "AlwaysTRUE" )
      wire#w1
      "MappingLossGroup"()
      "QueryLossGroupFromLossReason"(group_id := "DB_DataHMI".LossGroupSelectId, tab_index := "DB_DataHMI".PageDataLossReason.PageCurrent)
   END_RUNG
   RUNG wire#w1
      { S7_Templates := "SrcType := UInt" } EQ_Contact(in1 := "DB_DataHMI".EventCheckLossGroup, in2 := 1)
      wire#w2
      "CheckCheckBoxAssign"(index_checkbox := "DB_DataHMI".LossGroupSelectId, array_check_box := "DB_DataHMI".CheckboxLossGroup)
   END_RUNG
   RUNG wire#w2
      Move(in := 2, out1 => "DB_DataHMI".EventCheckLossGroup)
   END_RUNG
   RUNG wire#w2
      Move(in := 0, out1 => "DB_DataHMI".LossReasonSelectId)
   END_RUNG
   RUNG wire#w1
      { S7_Templates := "SrcType := UInt" } EQ_Contact(in1 := "DB_DataHMI".EventCheckLossReason, in2 := 1)
      wire#w3
      "CheckCheckBoxAssign"(index_checkbox := "DB_DataHMI".LossReasonSelectId, array_check_box := "DB_DataHMI".CheckboxLossReason)
   END_RUNG
   RUNG wire#w3
      Contact( "Tag_11" )
      Move(in := 2, out1 => "DB_DataHMI".EventCheckLossReason)
   END_RUNG
   // the same network as SCL:
   #_w2 := "AlwaysTRUE";
   "MappingLossGroup"(EN := "AlwaysTRUE", ENO => #_w1);
   IF #_w1 THEN
       "QueryLossGroupFromLossReason"(group_id := "DB_DataHMI".LossGroupSelectId,
                               tab_index := "DB_DataHMI".PageDataLossReason.PageCurrent);
   END_IF;
   #_w3 := #_w2 AND ("DB_DataHMI".EventCheckLossGroup = 1);
   IF #_w3 THEN
       "CheckCheckBoxAssign"(index_checkbox := "DB_DataHMI".LossGroupSelectId,
                             array_check_box := "DB_DataHMI".CheckboxLossGroup);
       "DB_DataHMI".EventCheckLossGroup := 2;
       "DB_DataHMI".LossReasonSelectId := 0;
   END_IF;
   #_w4 := #_w2 AND ("DB_DataHMI".EventCheckLossReason = 1);
   IF #_w4 THEN
       "CheckCheckBoxAssign"(index_checkbox := "DB_DataHMI".LossReasonSelectId,
                             array_check_box := "DB_DataHMI".CheckboxLossReason);
   END_IF;
   IF #_w4 AND "Tag_11" THEN "DB_DataHMI".EventCheckLossReason := 2; END_IF;
END_REGION

REGION Network 12 (SCL): Move Giá trị Loss group và loss reason
   #loss_group_id_temp := 0;
   IF "DB_DataHMI".LossReasonSelectId>=1 AND "DB_DataHMI".LossReasonSelectId<=10 THEN
       "DB_DataHMI".TextLossReasonAssignLossCurrent := "DB_DataHMI".LossDescriptionHmiDTO["DB_DataHMI".LossReasonSelectId].description;
       #loss_group_id_temp := "DB_DataHMI".LossDescriptionHmiDTO["DB_DataHMI".LossReasonSelectId].group_id;
   ELSE
       "DB_DataHMI".TextLossReasonAssignLossCurrent :='';
   END_IF;


   IF "DB_DataHMI".LossGroupSelectId=0 AND #loss_group_id_temp=0 THEN
       "DB_DataHMI".TextLossGroupAssignLossCurrent := 'All';
   ELSIF "DB_DataHMI".LossGroupSelectId=0 AND #loss_group_id_temp>=1 AND #loss_group_id_temp<=10 THEN
       "DB_DataHMI".TextLossGroupAssignLossCurrent := "DB_DataHMI".LossGroupHmiDTO[#loss_group_id_temp];
   ELSIF "DB_DataHMI".LossGroupSelectId>=1 AND "DB_DataHMI".LossGroupSelectId<=10 THEN
       "DB_DataHMI".TextLossGroupAssignLossCurrent := "DB_DataHMI".LossGroupHmiDTO["DB_DataHMI".LossGroupSelectId];
   ELSE
       "DB_DataHMI".TextLossGroupAssignLossCurrent := '';
   END_IF;

   //Clear nếu AssignLoss thành công hay bấm Cancel để để Default
   IF "DB_DataHMI".CancelAssignLoss=TRUE OR "DB_DataHMI".ActionAssignLossInShift=TRUE OR "DB_DataHMI".ActionAssignLossHistorical=TRUE THEN
       "DB_DataHMI".LossGroupSelectId := 0;
       //"DB_DataHMI".LossReasonSelectId := 0;
   END_IF;
END_REGION

REGION Network 13: Show Loss In Shift HMI
   RUNG wire#powerrail
      Contact( "AlwaysTRUE" )
      wire#w1
      { S7_Templates := "SrcType := UDInt" } LE_Contact(in1 := "DB_DataHMI".PageDataLossInShift.PageCurrent, in2 := 20)
      { S7_Templates := "SrcType := UDInt" } GT_Contact(in1 := "DB_DataHMI".PageDataLossInShift.PageCurrent, in2 := 0)
      wire#w2
      { S7_Templates := "SrcType := UDInt" } NE_Contact(in1 := "DB_DataHMI".PageDataLossInShift.PageCurrent, in2 := "DB_Machine".PageLossInShiftHmiPrevious)
      "ClearTableShowHMI"("1: table in shift, 2:table historical, 3: table spare part" := 1)
      "ClearBufferTempLossInShift"()
      Move(in := "DB_DataHMI".PageDataLossInShift.PageCurrent, out1 => "DB_Machine".PageLossInShiftHmiPrevious)
   END_RUNG
   RUNG wire#w2
      "SortBufferLossInShift"(page_current := "DB_DataHMI".PageDataLossInShift.PageCurrent, number_data_in_shift := "DB_DataHMI".PageDataLossInShift.TotalData)
   END_RUNG
   RUNG wire#w1
      { S7_Templates := "SrcType := UDInt" } LE_Contact(in1 := "DB_DataHMI".PageDataLossInShift.PageCurrent, in2 := 0)
      Move(in := 1, out1 => "DB_DataHMI".PageDataLossInShift.PageCurrent)
   END_RUNG
   // the same network as SCL:
   #_w1 := "AlwaysTRUE" AND ("DB_DataHMI".PageDataLossInShift.PageCurrent <= 20) AND ("DB_DataHMI".PageDataLossInShift.PageCurrent > 0);
   #_w3 := "AlwaysTRUE";
   "ClearTableShowHMI"(EN := #_w1 AND ("DB_DataHMI".PageDataLossInShift.PageCurrent <> "DB_Machine".PageLossInShiftHmiPrevious),
                       "1: table in shift, 2:table historical, 3: table spare part" := 1,
                       ENO => #_w2);
   "ClearBufferTempLossInShift"(EN := #_w2, ENO => #_w4);
   IF #_w4 THEN
       "DB_Machine".PageLossInShiftHmiPrevious := "DB_DataHMI".PageDataLossInShift.PageCurrent;
   END_IF;
   IF #_w1 THEN
       "SortBufferLossInShift"(page_current := "DB_DataHMI".PageDataLossInShift.PageCurrent,
                               number_data_in_shift := "DB_DataHMI".PageDataLossInShift.TotalData);
   END_IF;
   IF #_w3 AND ("DB_DataHMI".PageDataLossInShift.PageCurrent <= 0) THEN
       "DB_DataHMI".PageDataLossInShift.PageCurrent := 1;
   END_IF;
END_REGION

REGION Network 14: Show Loss Historical HMI
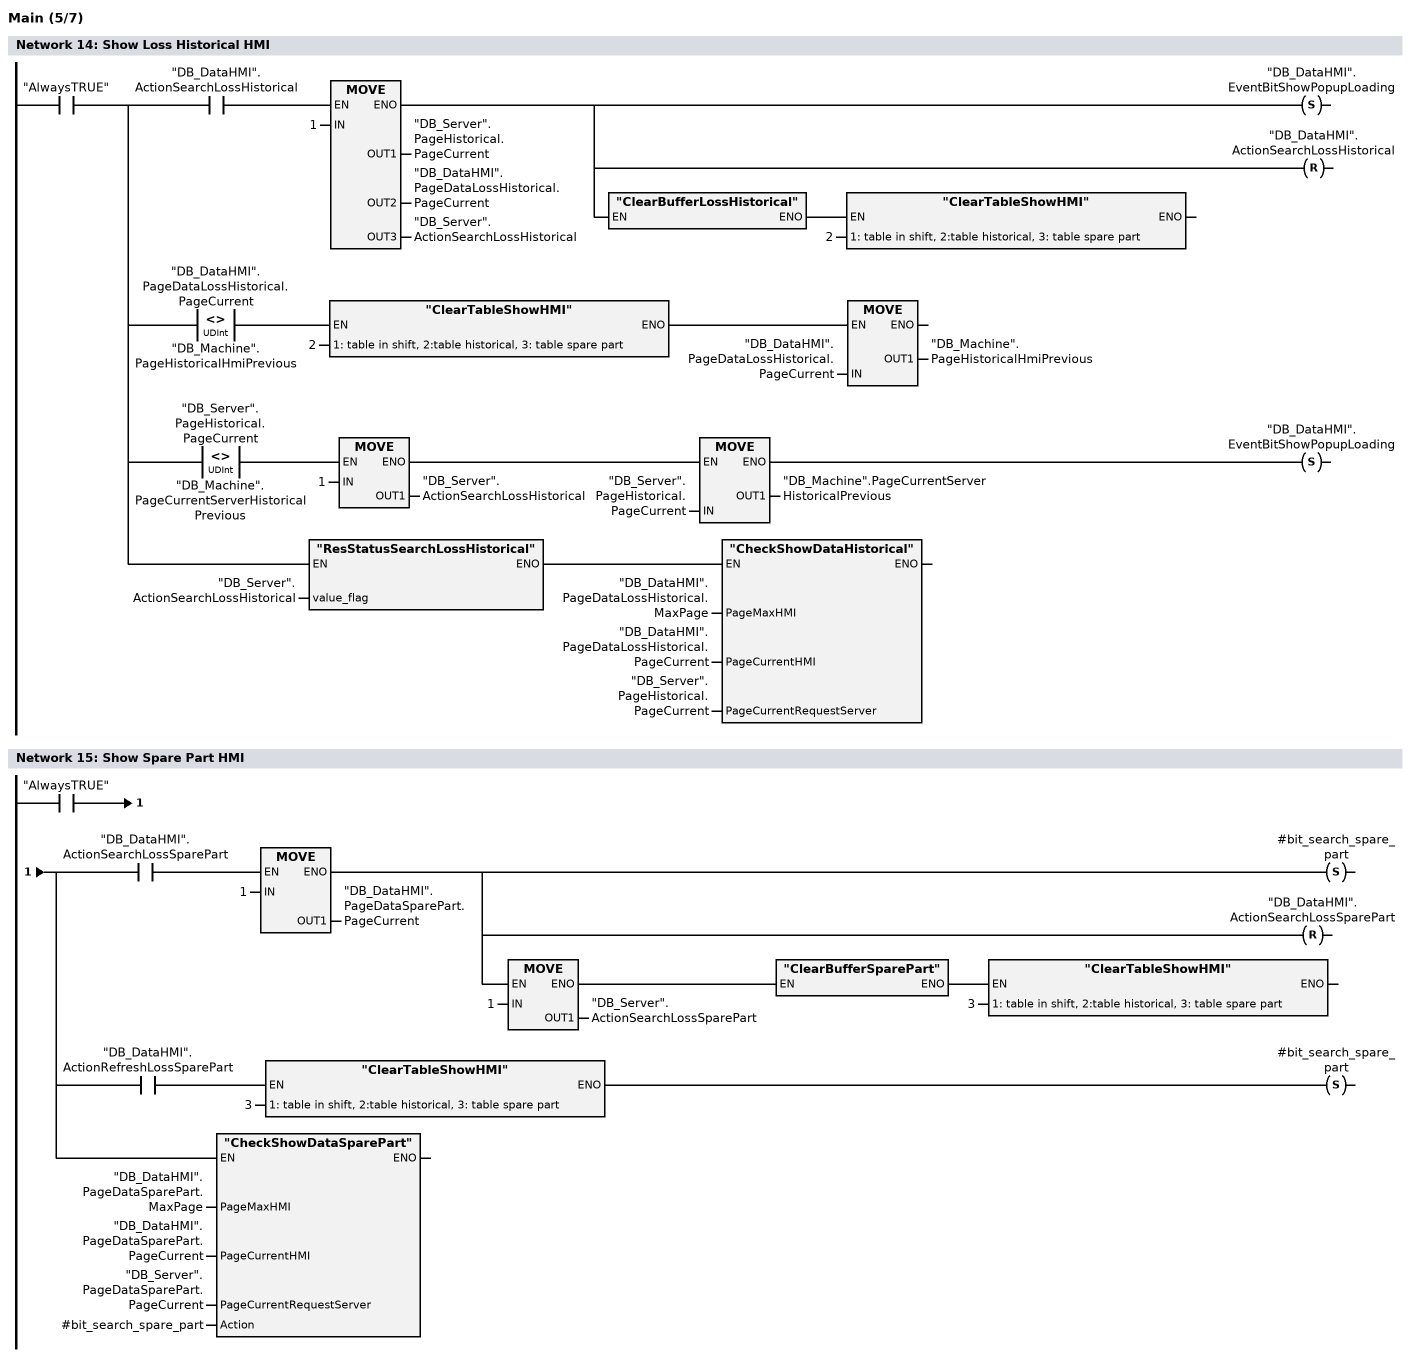
   RUNG wire#powerrail
      Contact( "AlwaysTRUE" )
      wire#w1
      Contact( "DB_DataHMI".ActionSearchLossHistorical )
      Move(in := 1, out1 => "DB_Server".PageHistorical.PageCurrent, out2 => "DB_DataHMI".PageDataLossHistorical.PageCurrent, out3 => "DB_Server".ActionSearchLossHistorical)
      wire#w2
      S_Coil( "DB_DataHMI".EventBitShowPopupLoading )
   END_RUNG
   RUNG wire#w2
      R_Coil( "DB_DataHMI".ActionSearchLossHistorical )
   END_RUNG
   RUNG wire#w2
      "ClearBufferLossHistorical"()
      "ClearTableShowHMI"("1: table in shift, 2:table historical, 3: table spare part" := 2)
   END_RUNG
   RUNG wire#w1
      { S7_Templates := "SrcType := UDInt" } NE_Contact(in1 := "DB_DataHMI".PageDataLossHistorical.PageCurrent, in2 := "DB_Machine".PageHistoricalHmiPrevious)
      "ClearTableShowHMI"("1: table in shift, 2:table historical, 3: table spare part" := 2)
      Move(in := "DB_DataHMI".PageDataLossHistorical.PageCurrent, out1 => "DB_Machine".PageHistoricalHmiPrevious)
   END_RUNG
   RUNG wire#w1
      { S7_Templates := "SrcType := UDInt" } NE_Contact(in1 := "DB_Server".PageHistorical.PageCurrent, in2 := "DB_Machine".PageCurrentServerHistoricalPrevious)
      Move(in := 1, out1 => "DB_Server".ActionSearchLossHistorical)
      Move(in := "DB_Server".PageHistorical.PageCurrent, out1 => "DB_Machine".PageCurrentServerHistoricalPrevious)
      S_Coil( "DB_DataHMI".EventBitShowPopupLoading )
   END_RUNG
   RUNG wire#w1
      "ResStatusSearchLossHistorical"(value_flag := "DB_Server".ActionSearchLossHistorical)
      "CheckShowDataHistorical"(PageMaxHMI := "DB_DataHMI".PageDataLossHistorical.MaxPage, PageCurrentHMI := "DB_DataHMI".PageDataLossHistorical.PageCurrent, PageCurrentRequestServer := "DB_Server".PageHistorical.PageCurrent)
   END_RUNG
   // the same network as SCL:
   IF "AlwaysTRUE" AND "DB_DataHMI".ActionSearchLossHistorical THEN
       "DB_Server".PageHistorical.PageCurrent := 1;
       "DB_DataHMI".PageDataLossHistorical.PageCurrent := 1;
       "DB_Server".ActionSearchLossHistorical := 1;
       "DB_DataHMI".EventBitShowPopupLoading := TRUE;
   END_IF;
   #_w1 := "AlwaysTRUE" AND "DB_DataHMI".ActionSearchLossHistorical;
   IF #_w1 THEN "DB_DataHMI".ActionSearchLossHistorical := FALSE; END_IF;
   #_w3 := "AlwaysTRUE";
   "ClearBufferLossHistorical"(EN := #_w1, ENO => #_w2);
   IF #_w2 THEN
       "ClearTableShowHMI"("1: table in shift, 2:table historical, 3: table spare part" := 2);
   END_IF;
   "ClearTableShowHMI"(EN := #_w3 AND ("DB_DataHMI".PageDataLossHistorical.PageCurrent <> "DB_Machine".PageHistoricalHmiPrevious),
                       "1: table in shift, 2:table historical, 3: table spare part" := 2,
                       ENO => #_w4);
   IF #_w4 THEN
       "DB_Machine".PageHistoricalHmiPrevious := "DB_DataHMI".PageDataLossHistorical.PageCurrent;
   END_IF;
   IF #_w3 AND ("DB_Server".PageHistorical.PageCurrent <> "DB_Machine".PageCurrentServerHistoricalPrevious) THEN
       "DB_Server".ActionSearchLossHistorical := 1;
   END_IF;
   #_w5 := #_w3 AND ("DB_Server".PageHistorical.PageCurrent <> "DB_Machine".PageCurrentServerHistoricalPrevious);
   IF #_w5 THEN
       "DB_Machine".PageCurrentServerHistoricalPrevious := "DB_Server".PageHistorical.PageCurrent;
       "DB_DataHMI".EventBitShowPopupLoading := TRUE;
   END_IF;
   "ResStatusSearchLossHistorical"(EN := #_w3,
                           value_flag := "DB_Server".ActionSearchLossHistorical,
                           ENO => #_w6);
   IF #_w6 THEN
       "CheckShowDataHistorical"(PageMaxHMI := "DB_DataHMI".PageDataLossHistorical.MaxPage,
                               PageCurrentHMI := "DB_DataHMI".PageDataLossHistorical.PageCurrent,
                               PageCurrentRequestServer := "DB_Server".PageHistorical.PageCurrent);
   END_IF;
END_REGION

REGION Network 15: Show Spare Part HMI
   RUNG wire#powerrail
      Contact( "AlwaysTRUE" )
      wire#w1
      Contact( "DB_DataHMI".ActionSearchLossSparePart )
      Move(in := 1, out1 => "DB_DataHMI".PageDataSparePart.PageCurrent)
      wire#w2
      S_Coil( #bit_search_spare_part )
   END_RUNG
   RUNG wire#w2
      R_Coil( "DB_DataHMI".ActionSearchLossSparePart )
   END_RUNG
   RUNG wire#w2
      Move(in := 1, out1 => "DB_Server".ActionSearchLossSparePart)
      "ClearBufferSparePart"()
      "ClearTableShowHMI"("1: table in shift, 2:table historical, 3: table spare part" := 3)
   END_RUNG
   RUNG wire#w1
      Contact( "DB_DataHMI".ActionRefreshLossSparePart )
      "ClearTableShowHMI"("1: table in shift, 2:table historical, 3: table spare part" := 3)
      S_Coil( #bit_search_spare_part )
   END_RUNG
   RUNG wire#w1
      "CheckShowDataSparePart"(PageMaxHMI := "DB_DataHMI".PageDataSparePart.MaxPage, PageCurrentHMI := "DB_DataHMI".PageDataSparePart.PageCurrent, PageCurrentRequestServer := "DB_Server".PageDataSparePart.PageCurrent, Action := #bit_search_spare_part)
   END_RUNG
   // the same network as SCL:
   IF "AlwaysTRUE" AND "DB_DataHMI".ActionSearchLossSparePart THEN
       "DB_DataHMI".PageDataSparePart.PageCurrent := 1;
       #bit_search_spare_part := TRUE;
   END_IF;
   #_w1 := "AlwaysTRUE" AND "DB_DataHMI".ActionSearchLossSparePart;
   IF #_w1 THEN
       "DB_DataHMI".ActionSearchLossSparePart := FALSE;
       "DB_Server".ActionSearchLossSparePart := 1;
   END_IF;
   #_w3 := "AlwaysTRUE";
   "ClearBufferSparePart"(EN := #_w1, ENO => #_w2);
   IF #_w2 THEN
       "ClearTableShowHMI"("1: table in shift, 2:table historical, 3: table spare part" := 3);
   END_IF;
   "ClearTableShowHMI"(EN := #_w3 AND "DB_DataHMI".ActionRefreshLossSparePart,
                       "1: table in shift, 2:table historical, 3: table spare part" := 3,
                       ENO => #_w4);
   IF #_w4 THEN #bit_search_spare_part := TRUE; END_IF;
   IF #_w3 THEN
       "CheckShowDataSparePart"(PageMaxHMI := "DB_DataHMI".PageDataSparePart.MaxPage,
                               PageCurrentHMI := "DB_DataHMI".PageDataSparePart.PageCurrent,
                               PageCurrentRequestServer := "DB_Server".PageDataSparePart.PageCurrent,
                               Action := #bit_search_spare_part);
   END_IF;
END_REGION

REGION Network 16: Move Infor Loss Assign To Page Assign
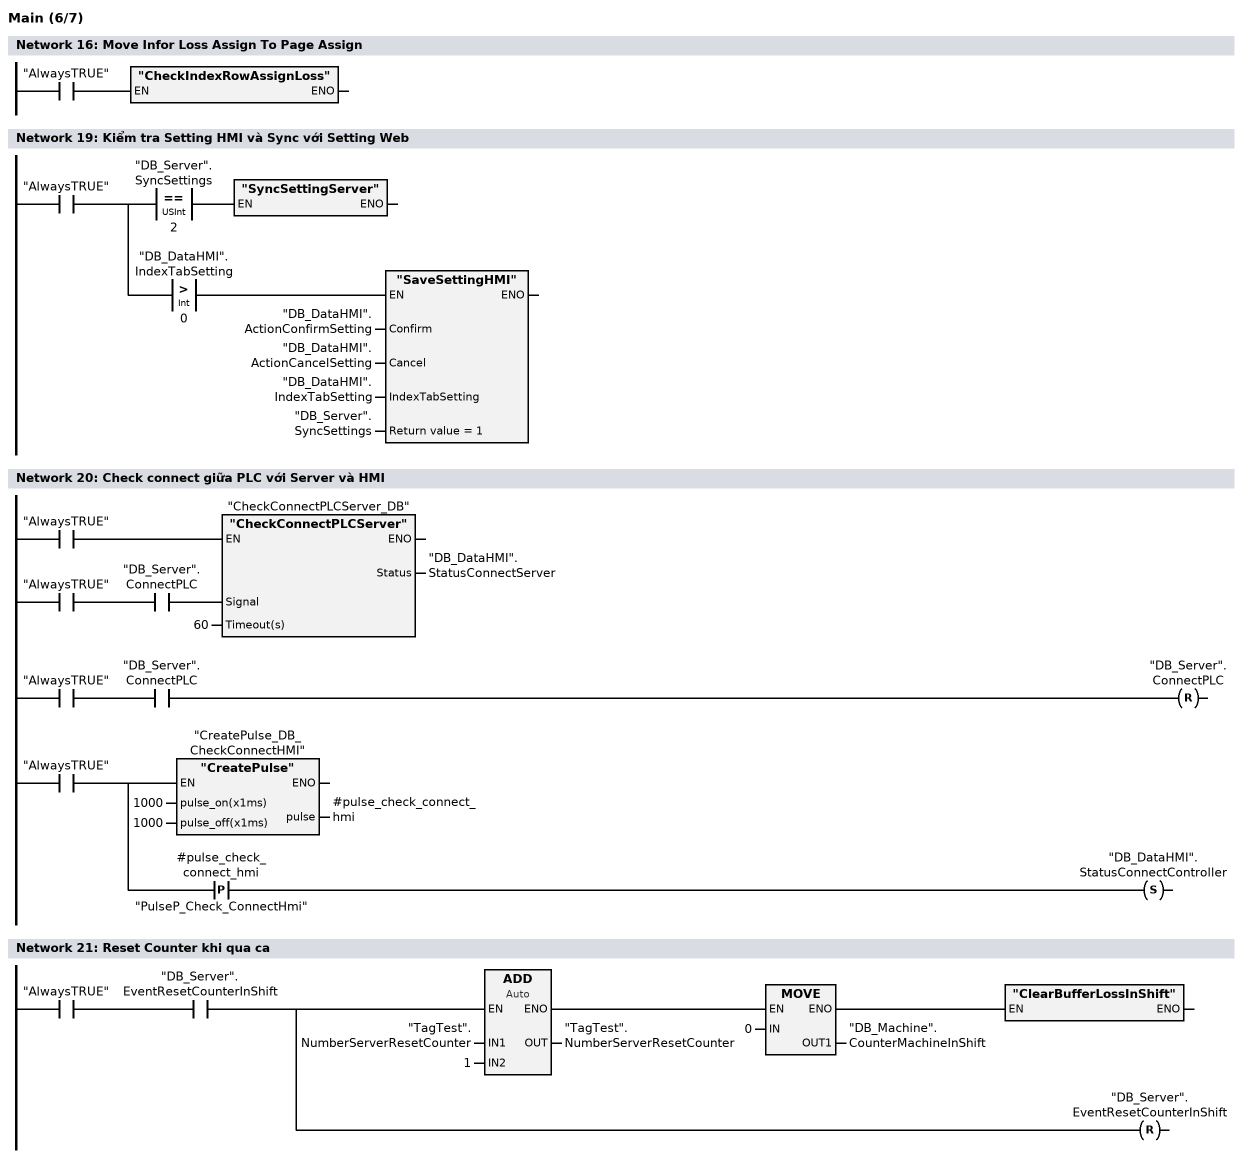
   RUNG wire#powerrail
      Contact( "AlwaysTRUE" )
      "CheckIndexRowAssignLoss"()
   END_RUNG
   // the same network as SCL:
   IF "AlwaysTRUE" THEN "CheckIndexRowAssignLoss"(); END_IF;
END_REGION

REGION Network 17 (SCL): Export data to HMI
   ////////////////////////////////// Monitor //////////////////////////////////
   //Mapping Input show display for HMI
   "DB_DataHMI".IO_Digital[1] := "M_Speed";
   "DB_DataHMI".IO_Digital[2] := "M_RunStop_Machine";
   "DB_DataHMI".IO_Digital[3] := "M_Xilanh_Push";
   "DB_DataHMI".IO_Digital[4] := "M_Pedal";
   "DB_DataHMI".IO_Digital[5] := "M_RunStop_Inverter";
   "DB_DataHMI".IO_Digital[6] := "Input 5 Spare";
   "DB_DataHMI".IO_Digital[7] := "Input 6 Spare";
   "DB_DataHMI".IO_Digital[8] := "Input 7 Spare";

   //////////////////////////////////Giá trị Realtime Sensor//////////////////////////////////
   //Blade Temperature
   "DB_DataHMI".BladeTemperature.AnalogActual := "M_Temperature";
   "DB_DataHMI".BladeTemperature."ValueActual(x100)" := "Analogs_DB".Temperature.CurrentDintValue;
   "DB_DataHMI".BladeTemperature."ValueActualContainOffset(x100)" := "Analogs_DB".Temperature.CurrentDintValue + "DataSetting".SettingBladeTemp."Offset(x100)";
   "CheckAlarmSensor"(Value:="DB_DataHMI".BladeTemperature."ValueActualContainOffset(x100)",
                      LowerSetting:="DataSetting".SettingBladeTemp."SettingLower(x100)",
                      UpperSetting:="DataSetting".SettingBladeTemp."SettingUpper(x100)",
                      Alarm=>"DB_DataHMI".BladeTemperature.Alarm);

   //Current
   "DB_DataHMI".Current.AnalogActual := "M_Current";
   IF "M_RunStop_Machine" = TRUE THEN
       "DB_DataHMI".Current."ValueActual(x100)" := "Analogs_DB".Current.CurrentDintValue;
       "DB_DataHMI".Current."ValueActualContainOffset(x100)" := "Analogs_DB".Current.CurrentDintValue + "DataSetting".SettingCurrent."Offset(x100)";
   ELSE
       "DB_DataHMI".Current."ValueActual(x100)" := 0;
       "DB_DataHMI".Current."ValueActualContainOffset(x100)" := 0;
   END_IF;

   "CheckAlarmSensor"(Value := "DB_DataHMI".Current."ValueActualContainOffset(x100)",
                      LowerSetting := "DataSetting".SettingCurrent."SettingLower(x100)",
                      UpperSetting := "DataSetting".SettingCurrent."SettingUpper(x100)",
                      Alarm => "DB_DataHMI".Current.Alarm);

   //Speed
   "CheckAlarmSensor"(Value := "DB_DataHMI".WheelSpeed."ValueActualContainOffset(x100)",
                      LowerSetting := "DataSetting".SettingWheelSpeed."SettingLower(x100)",
                      UpperSetting := "DataSetting".SettingWheelSpeed."SettingUpper(x100)",
                      Alarm => "DB_DataHMI".WheelSpeed.Alarm);

   //PresureOut
   "DB_DataHMI".PressureOut.AnalogActual := "M_Pressure Out";
   "DB_DataHMI"."ValuePressureOut_MPa(x100)" := "Analogs_DB".Pressure_OUT.CurrentDintValue;
   "DB_DataHMI".PressureOut."ValueActual(x100)" := REAL_TO_DINT("Analogs_DB".Pressure_OUT.CurrentRealValue * DINT_TO_REAL("DataSetting".SettingForceXilanh."CoefficientUnit(x100)"));
   "DB_DataHMI".PressureOut."ValueActualContainOffset(x100)" :="DB_DataHMI".PressureOut."ValueActual(x100)" + "DataSetting".SettingPresureOut."Offset(x100)";
   "CheckAlarmSensor"(Value := "DB_DataHMI".PressureOut."ValueActualContainOffset(x100)",
                      LowerSetting := "DataSetting".SettingPresureOut."SettingLower(x100)",
                      UpperSetting := "DataSetting".SettingPresureOut."SettingUpper(x100)",
                      Alarm => "DB_DataHMI".PressureOut.Alarm);


   ////////////////////////////////// Move Data vào vùng nhớ Chart /////////////////////////////////////////
   //Speed
   "DB_DataHMI".DataChartSpeed.Actual := ROUND_DINT(DINT_TO_REAL("DB_DataHMI".WheelSpeed."ValueActualContainOffset(x100)") / 100);
   "DB_DataHMI".DataChartSpeed.Min := ROUND_DINT(DINT_TO_REAL("DB_DataHMI".WheelSpeed.Common."SettingLower(x100)") / 100);
   "DB_DataHMI".DataChartSpeed.Max := ROUND_DINT(DINT_TO_REAL("DB_DataHMI".WheelSpeed.Common."SettingUpper(x100)") / 100);
   "CalculatorAxisYChart"(Actual := "DB_DataHMI".DataChartSpeed.Actual,
                          Min := "DB_DataHMI".DataChartSpeed.Min,
                          Max := "DB_DataHMI".DataChartSpeed.Max,
                          Min_AxisY => "DB_DataHMI".DataChartSpeed.AxisY_Min,
                          Max_AxisY => "DB_DataHMI".DataChartSpeed.AxisY_Max);

   //Current
   "DB_DataHMI".DataChartCurrent.Actual := ROUND_DINT(DINT_TO_REAL("DB_DataHMI".Current."ValueActualContainOffset(x100)") / 100);
   "DB_DataHMI".DataChartCurrent.Min := ROUND_DINT(DINT_TO_REAL("DB_DataHMI".Current.Common."SettingLower(x100)") / 100);
   "DB_DataHMI".DataChartCurrent.Max := ROUND_DINT(DINT_TO_REAL("DB_DataHMI".Current.Common."SettingUpper(x100)") / 100);
   "CalculatorAxisYChart"(Actual := "DB_DataHMI".DataChartCurrent.Actual,
                          Min := "DB_DataHMI".DataChartCurrent.Min,
                          Max := "DB_DataHMI".DataChartCurrent.Max,
                          Min_AxisY => "DB_DataHMI".DataChartCurrent.AxisY_Min,
                          Max_AxisY => "DB_DataHMI".DataChartCurrent.AxisY_Max);

   //BladeTemperature
   "DB_DataHMI".DataChartBladeTemperature.Actual := ROUND_DINT(DINT_TO_REAL("DB_DataHMI".BladeTemperature."ValueActualContainOffset(x100)") / 100);
   "DB_DataHMI".DataChartBladeTemperature.Min := ROUND_DINT(DINT_TO_REAL("DB_DataHMI".BladeTemperature.Common."SettingLower(x100)") / 100);
   "DB_DataHMI".DataChartBladeTemperature.Max := ROUND_DINT(DINT_TO_REAL("DB_DataHMI".BladeTemperature.Common."SettingUpper(x100)") / 100);
   "CalculatorAxisYChart"(Actual := "DB_DataHMI".DataChartBladeTemperature.Actual,
                          Min := "DB_DataHMI".DataChartBladeTemperature.Min,
                          Max := "DB_DataHMI".DataChartBladeTemperature.Max,
                          Min_AxisY => "DB_DataHMI".DataChartBladeTemperature.AxisY_Min,
                          Max_AxisY => "DB_DataHMI".DataChartBladeTemperature.AxisY_Max);

   //PressureOut
   "DB_DataHMI".DataChartPressureOut.Actual := ROUND_DINT(DINT_TO_REAL("DB_DataHMI".PressureOut."ValueActualContainOffset(x100)") / 10);
   "DB_DataHMI".DataChartPressureOut.Min := ROUND_DINT(DINT_TO_REAL("DB_DataHMI".PressureOut.Common."SettingLower(x100)") / 10);
   "DB_DataHMI".DataChartPressureOut.Max := ROUND_DINT(DINT_TO_REAL("DB_DataHMI".PressureOut.Common."SettingUpper(x100)") / 10);
   "CalculatorAxisYChart"(Actual := "DB_DataHMI".DataChartPressureOut.Actual,
                          Min := "DB_DataHMI".DataChartPressureOut.Min,
                          Max := "DB_DataHMI".DataChartPressureOut.Max,
                          Min_AxisY => "DB_DataHMI".DataChartPressureOut.AxisY_Min,
                          Max_AxisY => "DB_DataHMI".DataChartPressureOut.AxisY_Max);



   ///////////////////////////////////////////////////Status và Counter//////////////////////////////////////////////
   "DB_DataHMI".MachineStatus := "DB_Machine".MachineStatus;
   "DB_DataHMI".CounterCurrent := "DB_Machine".CounterMachineInShift;
   //Layer
   "DataSetting".TypeLayer := "DB_DataHMI".TypeLayer;


   /////////////////////////////////////////////////Số Loss trong ca/////////////////////////////////////////////////
   "DB_DataHMI".TotalDataInShift := "DB_Machine".NumberLossInShift;
   "DB_DataHMI".PageDataLossInShift.TotalData := "DB_Machine".NumberLossInShift;


   /////////////////////////////////////////////////Số Loss reason//////////////////////////////////////////////////
   "DB_DataHMI".PageDataLossReason.TotalData := "SettingsDB_LossDescription".number_loss_reason;


   /////////////////////////////////////////Lấy số Data Spare part  - Historical//////////////////////////////////////////////////
   "DB_DataHMI".PageDataSparePart.TotalData := "DB_Server".PageDataSparePart.TotalData;
   "DB_DataHMI".PageDataLossHistorical.TotalData := "DB_Server".PageHistorical.TotalData;


   ////////////////////////////////////////////Show TotalTime Page Historical///////////////////////////////////////
   "Cvt_Duration_to_String"("Time(ms)" := "DB_Server".TotalDurationPageHistorical,
                            ConvertTimeToStr => "DB_DataHMI".TotalTimeLossHistorical);


   /////////////////////////////////////////Lấy thông tin Setting//////////////////////////////////////////////////
   "DB_DataHMI".InforStation := "DataSetting".InforStation;



   //////////////////////Lấy thông tin Setting nếu có cờ flag///////////////////////
   IF "DB_DataHMI".BitReloadSettingToHMI THEN
       "MoveDataSettingToHmi"();
       "DB_DataHMI".BitReloadSettingToHMI := FALSE;
   END_IF;

   //////////////////////Lấy thông tin Setting move qua DB Analog///////////////////////
   "MoveDataSettingToBufferAnalog"();
END_REGION

REGION Network 18 (SCL): Sync Data Server - PLC
   //Dữ liệu từ Server gửi xuống
   "DataSetting".InforStation.Factory := "DB_Server".InforStation.Factory;
   "DataSetting".InforStation.Workshop := "DB_Server".InforStation.Workshop;
   "DataSetting".InforStation.LineName := "DB_Server".InforStation.LineName;
   "DataSetting".InforStation.MachineName := "DB_Server".InforStation.MachineName;

   // ////////////////////////////////////////////PLC -> Server/////////////////////////////////////////////////
   // //Value Sensor
   //Temp
   "DB_Server".SettingBladeTemp.AnalogCurrent := "DB_DataHMI".BladeTemperature.AnalogActual;
   "DB_Server".SettingBladeTemp."CurrentNotOffset(x100)" := "DB_DataHMI".BladeTemperature."ValueActual(x100)";
   "DB_Server".SettingBladeTemp."Current(x100)" := "DB_DataHMI".BladeTemperature."ValueActualContainOffset(x100)";
   "DB_Server".SettingBladeTemp.Alarm := "DB_DataHMI".BladeTemperature.Alarm;

   // //Current
   "DB_Server".SettingCurrent.AnalogCurrent := "DB_DataHMI".Current.AnalogActual;
   "DB_Server".SettingCurrent."CurrentNotOffset(x100)" := "DB_DataHMI".Current."ValueActual(x100)";
   "DB_Server".SettingCurrent."Current(x100)" := "DB_DataHMI".Current."ValueActualContainOffset(x100)";
   "DB_Server".SettingCurrent.Alarm := "DB_DataHMI".Current.Alarm;

   //Speed
   "DB_Server".SettingWheelSpeed.Infor."CurrentNotOffset(x100)" := "DB_DataHMI".WheelSpeed."ValueActual(x100)";
   "DB_Server".SettingWheelSpeed.Infor."Current(x100)" := "DB_DataHMI".WheelSpeed."ValueActualContainOffset(x100)";

   //Presure Out
   "DB_Server".SensorPresureOut.AnalogCurrent := "DB_DataHMI".PressureOut.AnalogActual;
   "DB_Server".SensorPresureOut."CurrentNotOffset(x100)" := "DB_DataHMI".PressureOut."ValueActual(x100)";
   "DB_Server".SensorPresureOut."Current(x100)" := "DB_DataHMI".PressureOut."ValueActualContainOffset(x100)";
   "DB_Server".SensorPresureOut.Alarm := "DB_DataHMI".PressureOut.Alarm;


   ///////////////////////////////Status và Counter///////////////////////////
   "DB_Server".MachineStatus := UINT_TO_SINT("DB_Machine".MachineStatus);
   "DB_Server".CounterMachineInShift := "DB_Machine".CounterMachineInShift;
   "DB_Server".CounterRaw := "DB_Machine".CounterRaw;

   "DB_Server".StartTimeStatusCurrent := "GLobalDB_LossManagementDB".current_status_machine.startTime;
   "DB_Server".EndTimeStatusCurrent := "GLobalDB_LossManagementDB".current_status_machine.endTime;
   "DB_Server".DurationStatusCurrent := "GLobalDB_LossManagementDB".current_status_machine.duration;

   /////////////////////////////Kiểu Layer ///////////////////////////
   "DB_Server".TypeLayer := "DB_DataHMI".TypeLayer;


   /////////////////////////////HMI yêu cầu lấy data từ Server////////////////////////////
   //Search Historical
   IF "DB_DataHMI".ActionSearchLossHistorical=TRUE THEN
       "DB_Server".SearchDataLossHistorical := "DB_DataHMI".SearchDataLoss;
       "DB_Server".ActionSearchLossHistorical := 1;
       "DB_DataHMI".ActionSearchLossHistorical := FALSE;
   END_IF;
   "ReturnPageFromTotalData"(total_data:="DB_Server".PageHistorical.TotalData,
                             data_per_page:=50,
                             total_page=>"DB_Server".PageHistorical.MaxPage);
   IF "DB_Server".PageHistorical.MaxPage>20 THEN
       "DB_Server".PageHistorical.MaxPage := 20;
   END_IF;


   //Reload Group ReasonLoss
   IF "DB_DataHMI".RequestLoadGroupReasonLoss = TRUE THEN
       "DB_Server".RequestServerWriteLossGroup_Reason := 1;
       "DB_DataHMI".RequestLoadGroupReasonLoss := FALSE;
   END_IF;
END_REGION

REGION Network 19: Kiểm tra Setting HMI và Sync với Setting Web
   RUNG wire#powerrail
      Contact( "AlwaysTRUE" )
      wire#w1
      { S7_Templates := "SrcType := USInt" } EQ_Contact(in1 := "DB_Server".SyncSettings, in2 := 2)
      "SyncSettingServer"()
   END_RUNG
   RUNG wire#w1
      { S7_Templates := "SrcType := Int" } GT_Contact(in1 := "DB_DataHMI".IndexTabSetting, in2 := 0)
      "SaveSettingHMI"(Confirm := "DB_DataHMI".ActionConfirmSetting, Cancel := "DB_DataHMI".ActionCancelSetting, IndexTabSetting := "DB_DataHMI".IndexTabSetting, "Return value = 1" := "DB_Server".SyncSettings)
   END_RUNG
   // the same network as SCL:
   #_w1 := "AlwaysTRUE";
   IF "AlwaysTRUE" AND ("DB_Server".SyncSettings = 2) THEN "SyncSettingServer"(); END_IF;
   IF #_w1 AND ("DB_DataHMI".IndexTabSetting > 0) THEN
       "SaveSettingHMI"(Confirm := "DB_DataHMI".ActionConfirmSetting,
                        Cancel := "DB_DataHMI".ActionCancelSetting,
                        IndexTabSetting := "DB_DataHMI".IndexTabSetting,
                        "Return value = 1" := "DB_Server".SyncSettings);
   END_IF;
END_REGION

